# B&R Automation Studio project BaseProject (part 2)

### TrackMod.vvm - PC/TrackModule/TrackMod.vvm
```iecst
VAR_CONFIG
	Cyclic#1.::gSampleTrak AT %Q.TrackModule::TrackInterface.SampleTrak; (*Insert your comment here...*)
	Cyclic#1.TrackModule::gTrackModule AT %Q.TrackModule::TrackInterface.ModulePml; (*Insert your comment here...*)
	Cyclic#1.TrackModule::gAlarmXCore_TrackModule AT %Q.TrackModule::TrackInterface.AlarmCore; (*Insert your comment here...*)
	Cyclic#1.TrackModule::gRecipeXml_TrackModule AT %Q.TrackModule::TrackInterface.RecipeCore; (*Insert your comment here...*)
END_VAR
```

### TrakALM.mpalarmxcore - PC/TrackModule/mappServices/TrakALM.mpalarmxcore
```
Element gAlarmXCore_TrackModule (Type=mpalarmxcore)
  mapp.AlarmX.Core:
    Mapping:
      [0]:
        Alarm = Inf*
        [0] = Aggregate
          Name = TrakModuleInfo
      [1]:
        Alarm = Warn*
        [0] = Aggregate
          Name = TrakModuleWarning
      [2]:
        Alarm = Alrm*
        [0] = Aggregate
          Name = TrakModuleAlarm
    Default:
      [0] = Reaction
        Name = TrakTest
      [1] = Remain
  mapp.AlarmX.Core.Configuration:
    [0]:
      Name = Alrm_ErrorStop
      Message = {$TrakAssembly/TrakErrorStop}
      Code = 1000
      Behavior = DiscreteValueMonitoring
        Monitoring:
          MonitoredPV = TrakModule::AsmSampleT:fbAsmReadStatus.AssemblyErrorStop
          TriggerValues:
            [0] = TRUE
    [1]:
      Name = Inf_PowerOn
      Message = {$Assembly/Info/TrakPowerOn}
      Behavior = DiscreteValueMonitoring
        Monitoring:
          MonitoredPV = TrakModule::AsmSampleT:fbAsmReadInfo.AssemblyInfo.PowerOn
          TriggerValues:
            [0] = TRUE
    [2]:
      Name = Inf_ModuleTest
      Message = {$TrakAssembly/LocalTrakModuleInfo}
      Severity = 0
      Behavior = DiscreteValueMonitoring
        Monitoring:
          MonitoredPV = TrakModule::AsmAlarm:TriggerTestInformation
          TriggerValues:
            [0] = TRUE
    [3]:
      Name = Warn_ModuleTest
      Message = {$TrakAssembly/LocalTrakModuleWarning}
      Code = 100
      Severity = 50
      Behavior = DiscreteValueMonitoring
        Monitoring:
          MonitoredPV = TrakModule::AsmAlarm:TriggerTestWarning
          TriggerValues:
            [0] = TRUE
    [4]:
      Name = Alrm_ModuleTest
      Message = {$TrakAssembly/LocalTrakModuleAlarm}
      Code = 1000
      Severity = 100
      Behavior = DiscreteValueMonitoring
        Monitoring:
          MonitoredPV = TrakModule::AsmAlarm:TriggerTestAlarm
          TriggerValues:
            [0] = TRUE
    [5]:
      Name = TrakModuleInfo
      Message = {$TrakAssembly/Module.Info}
      AdditionalInformation1 = trakAlarmContent
    [6]:
      Name = TrakModuleWarning
      Message = {$TrakAssembly/Module.Warning}
      Code = 100
      AdditionalInformation1 = trakAlarmContent
    [7]:
      Name = TrakModuleAlarm
      Message = {$TrakAssembly/Module.Alarm}
      Code = 1000
      AdditionalInformation1 = trakAlarmContent
  mapp.AlarmX.Core.Snippets:
    [0]:
      Key = ModuleName
      Value:
        PV = TrakModule::ModuleName
  mapp.AlarmX.Core.Categories:
    [0]:
      Name = Information
      SourceProperty:
        Severity = 0..99
    [1]:
      Name = Warning
      SourceProperty:
        Severity = 100..199
    [2]:
      Name = Alarm
      SourceProperty:
        Severity = 1000..1199
```

### TrakMod.vvm - PC/TrakMod/TrakMod.vvm
```iecst
VAR_CONFIG
	Cyclic#1.::gSampleTrak AT %Q.Cyclic#1.TrakMod::TrakInterface.SampleTrak; (*Insert your comment here...*)
	Cyclic#1.TrakMod::gTrakModule AT %Q.Cyclic#1.TrakMod::TrakInterface.ModulePml; (*Insert your comment here...*)
	Cyclic#1.TrakMod::gAlarmXCore_TrakModule AT %Q.Cyclic#1.TrakMod::TrakInterface.AlarmCore; (*Insert your comment here...*)
	Cyclic#1.TrakMod::gRecipeXml_TrakModule AT %Q.Cyclic#1.TrakMod::TrakInterface.RecipeCore; (*Insert your comment here...*)
	Cyclic#1.::gSampleTrak_SectorTrakAll AT %Q.Cyclic#1.TrakMod::TrakInterface.SectorTrakAll; (*Insert your comment here...*)
	Cyclic#1.::gSampleTrak_SectorTrakB AT %Q.Cyclic#1.TrakMod::TrakInterface.SectorTrakB; (*Insert your comment here...*)
	Cyclic#1.::gSampleTrak_SectorTrakA AT %Q.Cyclic#1.TrakMod::TrakInterface.SectorTrakA; (*Insert your comment here...*)
END_VAR
```

### TrakALM.mpalarmxcore - PC/TrakMod/mappServices/TrakALM.mpalarmxcore
```
Element gAlarmXCore_TrakModule (Type=mpalarmxcore)
  mapp.AlarmX.Core:
    Mapping:
      [0]:
        Alarm = Inf*
        [0] = Aggregate
          Name = TrakModuleInfo
      [1]:
        Alarm = Warn*
        [0] = Aggregate
          Name = TrakModuleWarning
      [2]:
        Alarm = Alrm*
        [0] = Aggregate
          Name = TrakModuleAlarm
    Default:
      [0] = Remain
      [1] = Reaction
        Name = TrakTest
  mapp.AlarmX.Core.Configuration:
    [0]:
      Name = Alrm_ErrorStop
      Message = {$TrakAssembly/TrakErrorStop}
      Code = 1000
      Behavior = DiscreteValueMonitoring
        Monitoring:
          MonitoredPV = TrakMod::AsmSampleT:fbAsmReadStatus.AssemblyErrorStop
          TriggerValues:
            [0] = TRUE
    [1]:
      Name = Inf_PowerOn
      Message = {$TrakAssembly/TrakPowerOn}
      Behavior = DiscreteValueMonitoring
        Monitoring:
          MonitoredPV = TrakMod::AsmSampleT:fbAsmReadInfo.AssemblyInfo.PowerOn
          TriggerValues:
            [0] = TRUE
    [2]:
      Name = Inf_ModuleTest
      Message = {$TrakAssembly/LocalTrakModuleInfo}
      Severity = 0
      Behavior = DiscreteValueMonitoring
        Monitoring:
          MonitoredPV = TrakMod::AsmAlarm:TriggerTestInformation
          TriggerValues:
            [0] = TRUE
    [3]:
      Name = Warn_ModuleTest
      Message = {$TrakAssembly/LocalTrakModuleWarning}
      Code = 100
      Severity = 50
      Behavior = DiscreteValueMonitoring
        Monitoring:
          MonitoredPV = TrakMod::AsmAlarm:TriggerTestWarning
          TriggerValues:
            [0] = TRUE
    [4]:
      Name = Alrm_ModuleTest
      Message = {$TrakAssembly/LocalTrakModuleAlarm}
      Code = 1000
      Severity = 100
      Behavior = DiscreteValueMonitoring
        Monitoring:
          MonitoredPV = TrakMod::AsmAlarm:TriggerTestAlarm
          TriggerValues:
            [0] = TRUE
    [5]:
      Name = TrakModuleInfo
      Message = {$TrakAssembly/Module.Info}
      AdditionalInformation1 = trakAlarmContent
    [6]:
      Name = TrakModuleWarning
      Message = {$TrakAssembly/Module.Warning}
      Code = 100
      AdditionalInformation1 = trakAlarmContent
    [7]:
      Name = TrakModuleAlarm
      Message = {$TrakAssembly/Module.Alarm}
      Code = 1000
      AdditionalInformation1 = trakAlarmContent
  mapp.AlarmX.Core.Snippets:
    [0]:
      Key = ModuleName
      Value:
        PV = TrakMod::ModuleName
  mapp.AlarmX.Core.Categories:
    [0]:
      Name = Information
      SourceProperty:
        Severity = 0..99
    [1]:
      Name = Warning
      SourceProperty:
        Severity = 100..199
    [2]:
      Name = Alarm
      SourceProperty:
        Severity = 1000..1199
```

### TrakCFG.mprecipexml - PC/TrakMod/mappServices/TrakCFG.mprecipexml
```
Element gRecipeXml_TrakModule (Type=mprecipexml)
  Alarms = MpAlarmX
```

### TrakPML.mppackmlmodule - PC/TrakMod/mappServices/TrakPML.mppackmlmodule
```
Element gTrakModule (Type=mppackmlmodule)
  Module:
    Name = TrakAssembly
    Parent:
      Parent = gMainModule
      Activation = 0
```

### TrakModule.vvm - PC/TrakModule/TrakModule.vvm
```iecst
VAR_CONFIG
	Cyclic#1.::gSampleTrak AT %Q.TrakModule::TrakInterface.SampleTrak; (*Insert your comment here...*)
	Cyclic#1.TrakModule::gTrakModule AT %Q.TrakModule::TrakInterface.ModulePml; (*Insert your comment here...*)
	Cyclic#1.TrakModule::gAlarmXCore_TrakModule AT %Q.TrakModule::TrakInterface.AlarmCore; (*Insert your comment here...*)
	Cyclic#1.TrakModule::gRecipeXml_TrackModule AT %Q.TrakModule::TrakInterface.RecipeCore; (*Insert your comment here...*)
END_VAR
```

### TrakALM.mpalarmxcore - PC/TrakModule/mappServices/TrakALM.mpalarmxcore
```
Element gAlarmXCore_TrakModule (Type=mpalarmxcore)
  mapp.AlarmX.Core:
    Mapping:
      [0]:
        Alarm = Inf*
        [0] = Aggregate
          Name = TrakModuleInfo
      [1]:
        Alarm = Warn*
        [0] = Aggregate
          Name = TrakModuleWarning
      [2]:
        Alarm = Alrm*
        [0] = Aggregate
          Name = TrakModuleAlarm
    Default:
      [0] = Reaction
        Name = TrakTest
      [1] = Remain
  mapp.AlarmX.Core.Configuration:
    [0]:
      Name = Alrm_ErrorStop
      Message = {$TrakAssembly/TrakErrorStop}
      Code = 1000
      Behavior = DiscreteValueMonitoring
        Monitoring:
          MonitoredPV = TrakModule::AsmSampleT:fbAsmReadStatus.AssemblyErrorStop
          TriggerValues:
            [0] = TRUE
    [1]:
      Name = Inf_PowerOn
      Message = {$Assembly/Info/TrakPowerOn}
      Behavior = DiscreteValueMonitoring
        Monitoring:
          MonitoredPV = TrakModule::AsmSampleT:fbAsmReadInfo.AssemblyInfo.PowerOn
          TriggerValues:
            [0] = TRUE
    [2]:
      Name = Inf_ModuleTest
      Message = {$TrakAssembly/LocalTrakModuleInfo}
      Severity = 0
      Behavior = DiscreteValueMonitoring
        Monitoring:
          MonitoredPV = TrakModule::AsmAlarm:TriggerTestInformation
          TriggerValues:
            [0] = TRUE
    [3]:
      Name = Warn_ModuleTest
      Message = {$TrakAssembly/LocalTrakModuleWarning}
      Code = 100
      Severity = 50
      Behavior = DiscreteValueMonitoring
        Monitoring:
          MonitoredPV = TrakModule::AsmAlarm:TriggerTestWarning
          TriggerValues:
            [0] = TRUE
    [4]:
      Name = Alrm_ModuleTest
      Message = {$TrakAssembly/LocalTrakModuleAlarm}
      Code = 1000
      Severity = 100
      Behavior = DiscreteValueMonitoring
        Monitoring:
          MonitoredPV = TrakModule::AsmAlarm:TriggerTestAlarm
          TriggerValues:
            [0] = TRUE
    [5]:
      Name = TrakModuleInfo
      Message = {$TrakAssembly/Module.Info}
      AdditionalInformation1 = trakAlarmContent
    [6]:
      Name = TrakModuleWarning
      Message = {$TrakAssembly/Module.Warning}
      Code = 100
      AdditionalInformation1 = trakAlarmContent
    [7]:
      Name = TrakModuleAlarm
      Message = {$TrakAssembly/Module.Alarm}
      Code = 1000
      AdditionalInformation1 = trakAlarmContent
  mapp.AlarmX.Core.Snippets:
    [0]:
      Key = ModuleName
      Value:
        PV = TrakModule::ModuleName
  mapp.AlarmX.Core.Categories:
    [0]:
      Name = Information
      SourceProperty:
        Severity = 0..99
    [1]:
      Name = Warning
      SourceProperty:
        Severity = 100..199
    [2]:
      Name = Alarm
      SourceProperty:
        Severity = 1000..1199
```

### TrakCFG.mprecipexml - PC/TrakModule/mappServices/TrakCFG.mprecipexml
```
Element gRecipeXml_TrackModule (Type=mprecipexml)
  Alarms = MpAlarmX
```

### LoggerCFG.mappmotioncfg - PC/mappMotion/LoggerCFG.mappmotioncfg
```
Element MappMotionConfiguration (Type=mappmotioncfg)
  Logger:
    SelectiveLogging = Used
      AdministrativeCommands = Selective
      MovementCommands = Selective
      InformationalCommands = Selective
```

### AsmCfg.assembly - PC/mappMotion/TrakConfig/AsmCfg.assembly
```
Element gSampleTrak (Type=assembly)
  Tracks:
    TrackSeparation = 0.030
    Track[1]:
      Segments:
        SegmentRef[1] = ::gSeg_A_1
        SegmentRef[2] = ::gSeg_A_2
        SegmentRef[3] = ::gSeg_A_3
        SegmentRef[4] = ::gSeg_A_4
        SegmentRef[5] = ::gSeg_A_5
        SegmentRef[6] = ::gSeg_A_6
        SegmentRef[7] = ::gSeg_A_7
        SegmentRef[8] = ::gSeg_A_8
        SegmentRef[9] = ::gSeg_A_9
        SegmentRef[10] = ::gSeg_A_10
        SegmentRef[11] = ::gSeg_A_11
        SegmentRef[12] = ::gSeg_A_12
      Position = Absolute
        SegmentRef = ::gSeg_A_1
        SegmentCountDirection = RightToLeft
        Translation:
          X = 0.0
          Y = 0.0
          Z = 0.0
        Orientation:
          Angle1 = 0.0
          Angle2 = 0.0
          Angle3 = 180
  CommonSegmentSettings:
    SegmentSimulationOnPLC = Off
    StopReaction = InductionHalt
    SpeedFilter = NotUsed
    ControllerParameters:
      DefaultParameter:
        Controller:
          Position:
            ProportionalGain = 200
          Speed:
            ProportionalGain = 80
            IntegrationTime = 0.0
          FeedForward:
            TotalMass = 1
            ForcePositive = 0.0
            ForceNegative = 0.0
            SpeedForceFactor = 0.0
            ForceLoad = 0.0
        MovementErrorLimits:
          PositionError = 0.001
          VelocityError = 0.05
      AdditionalParameterSets = NotUsed
    ScopeOfErrorReaction = Assembly
    ShuttleIdentificationTime = 0
  Shuttles:
    MaxShuttleCount = 150
    DistanceReserve:
      Collision = 0.002
      ErrorStop = 0.006
    ShuttleStereotypes:
      ShuttleStRef[1] = gSampleShuttle
    MagnetPlateConfigurations:
      ShuttleType[1] = 8F1SA.100.xxxxxx-x
    CollisionAvoidance:
      Strategy = Constant
      MaximumModelDimensions:
        Length:
          ExtentToFront = 0.025
          ExtentToBack = 0.025
        Width:
          Width = 0.040
  AssemblyFeatures:
    AssemblyFeatureRef[1] = SampleTrak_AutoAttach
    AssemblyFeatureRef[2] = SampleTrak_LocalLimits
    AssemblyFeatureRef[3] = SampleTrak_SimShuttle
  Visualization:
    MonitoringPv = gSampleTrakMon
    ProcessingTaskClass = 1
```

### AsmFeatCfg.assemblyfeature - PC/mappMotion/TrakConfig/AsmFeatCfg.assemblyfeature
```
Element SampleTrak_AutoAttach (Type=assemblyfeature)
  Type = ShtSectorAutoAttach
    Priority[1]:
      SectorRef = SampleTrak_SectorTrackA
      Orientation = KeepSegment
Element SampleTrak_LocalLimits (Type=assemblyfeature)
  Type = LocalLimits
    LocalLimit[1]:
      Location:
        SectorRef = SampleTrak_SectorTrackA
      MotionLimits:
        Velocity = Basic
          Velocity = 3
        Acceleration = Basic
          Acceleration = 10
Element SampleTrak_SimShuttle (Type=assemblyfeature)
  Type = InitShuttleSim
    InitShuttleSim[1]:
      SectorRef = SampleTrak_SectorTrackA
      Orientation = Positive
      ShuttleDefinition = ShuttleSetDefinition
        StartPosition = 0.0
        NumberOfShuttles = 10
        DistnaceBetweenShuttles = 100
Element SampleTrak_AsmPwr_STO1 (Type=assemblyfeature)
  Type = ExcludeFromAssembly
    Exclusion = AsmPowerOn
      SegmentRef[1] = ::Seg_A_1
      SegmentRef[2] = ::Seg_A_2
Element SampleTrak_AsmPwr_STO2 (Type=assemblyfeature)
  Type = ExcludeFromAssembly
    Exclusion = AsmPowerOn
      SegmentRef[1] = ::Seg_A_3
      SegmentRef[2] = ::Seg_A_4
```

### SectorCfg.sector - PC/mappMotion/TrakConfig/SectorCfg.sector
```
Element gSampleTrak_SectorTrakA (Type=sector)
  Type = Composed
    StartSegment:
      SegmentRef = ::gSeg_A_1
    IntermediateSegments:
      SegmentRef[1] = ::gSeg_A_2
      SegmentRef[2] = ::gSeg_A_3
      SegmentRef[3] = ::gSeg_A_4
      SegmentRef[4] = ::gSeg_A_5
      SegmentRef[5] = ::gSeg_A_6
      SegmentRef[6] = ::gSeg_A_7
      SegmentRef[7] = ::gSeg_A_8
      SegmentRef[8] = ::gSeg_A_9
      SegmentRef[9] = ::gSeg_A_10
      SegmentRef[10] = ::gSeg_A_11
    EndSegment:
      SegmentRef = ::gSeg_A_12
      PositionRelativeTo = FromEnd
```

### ShuttleCfg.shuttlestereotype - PC/mappMotion/TrakConfig/ShuttleCfg.shuttlestereotype
```
Element SampleShuttle (Type=shuttlestereotype)
  MeasurementUnit = 5067858
  MeasurementResolution = 0.00001
  MovementLimits = Internal
    VelocityIsReadOnly = 0
    Velocity:
      Velocity = 4
    AccelerationIsReadOnly = 0
    Acceleration:
      Acceleration = 40
    DecelerationIsReadOnly = 0
    Deceleration:
      Deceleration = 40
  JerkFilter = Used
    JerkTime = 0.02
  UserData:
    Size = 12
```

### MainAlrCfg.mpalarmxcore - PC/mappServices/Alarm/MainAlrCfg.mpalarmxcore
```
Element gAlarmXCore (Type=mpalarmxcore)
  mapp.AlarmX.Core:
    Mapping:
      [0]
  mapp.AlarmX.Core.Configuration:
    [0]:
      Name = MainTestAlarm
      Message = This is just a test for main
      Behavior = DiscreteValueMonitoring
        Monitoring:
          MonitoredPV = ::TSMAlarm:TriggerTestAlarm
          TriggerValues:
            [0] = TRUE
```

### AuditCfg.mpaudittrail - PC/mappServices/Diagnostic/AuditCfg.mpaudittrail
```
Element gAuditTrail (Type=mpaudittrail)
  Audit:
    Events:
      [0] = 18
    TextSource:
      OutputFormat = {&typ} | {&msg} | {&cmt}
  Alarms = MpAlarmX
```

### MachCfg.mprecipexml - PC/mappServices/MachineConfig/MachCfg.mprecipexml
```
Element gRecipeXml (Type=mprecipexml)
  Alarms = MpAlarmX
```

### Main.mppackmlmodule - PC/mappServices/Operation/Main.mppackmlmodule
```
Element gMainModule (Type=mppackmlmodule)
  Module:
    Parent = 1
      Unit = gPackMLCore
      Activation = 0
```

## Logical view

Binary libraries used (declarations not repeated): operator, runtime, astime, AsIecCon, AsZip, FileIO, sys_lib, snprintf 1.10.2, brdkSTR, ArEventLog, AsHttp, AsIODiag, AsBrStr, standard, asstring, McBase 5.15.1, McAcpPar 5.15.1, McAxGroup 5.15.1, McAcpAx 5.15.1, McAxis 5.15.1, McPathGen 5.15.1, McProgInt 5.15.1, McAcpTrak 5.15.1, MpRobotics 5.15.1, MpAxis 5.15.1, MpBase 5.15.0, MpCom 5.14.0, MpPackML 5.15.0, MpFile 5.15.0, MpAudit 5.15.0, MpRecipe 5.15.0, MpAlarmX 5.15.0, CoTrace 5.15.0, MpServer 5.15.0

### Global.typ - Global data types
```iecst
TYPE
	ShuttleUserDataType : 	STRUCT  (*Shuttle data type definition - application specific*)
		ID : UINT; (*Shuttle ID assigned during homing*)
	END_STRUCT;
	SubroutineSequenceType : 	STRUCT  (*Subroutine sequence structure for a module*)
		Cmd : SubroutineSequenceCommandType; (*Subroutine commands (inputs)*)
		Status : SubroutineSequenceStatusType; (*Subroutine statuses (outputs)*)
	END_STRUCT;
	SubroutineSequenceCommandType : 	STRUCT  (*Subroutine seguence command variables*)
		Start : BOOL; (*Initiate the subroutine execution when the status reports ready*)
		Stop : BOOL; (*If the main routine is no longer in a proper state to execute the subroutine, stop the subroutine*)
		ErrorReset : BOOL; (*Command to reset the subroutine if in error*)
	END_STRUCT;
	SubroutineSequenceStatusType : 	STRUCT  (*Subroutine segeuqnce status variables*)
		Ready : BOOL; (*The subroutine is ready to start*)
		Complete : BOOL; (*The subroutine has complete and will wait for the reset of the start command*)
		Error : BOOL; (*The subroutine is in error and needs to be reset*)
	END_STRUCT;
	CyclicSubroutineType : 	STRUCT  (*Cyclic subroutine structure definition for a module*)
		Cmd : CyclicSubroutineCommandType; (*Cyclic subroutine command structure*)
		Status : CyclicSubroutineStatusType; (*Cyclic subroutine status structure*)
	END_STRUCT;
	CyclicSubroutineCommandType : 	STRUCT  (*Cyclic subroutine command structure definition*)
		Activate : BOOL; (*Activate the subroutine cyclic operation*)
		ErrorReset : BOOL; (*Reset the subroutine when in error*)
	END_STRUCT;
	CyclicSubroutineStatusType : 	STRUCT  (*Cyclic subroutine status structure definition*)
		Ready : BOOL; (*The subroutine cyclic operation is ready to begin*)
		Active : BOOL; (*The subroutine is activated and running*)
		Error : BOOL; (*The subroutine is in error*)
	END_STRUCT;
END_TYPE

(*Trak Data Datatypes*)
```

### Global.var - Global variables
```iecst
VAR
	gTrakData : TrkDiagStatusType;
END_VAR
```

### Package Logical/Libraries - Global libraries

### Library Logical/Libraries/TrBase (IEC) - AddOn Trak library for types and variable definitions

#### TrBase.typ - Exported data types
```iecst
(*Assembly States*)

TYPE
	TrBaseAsmStateEnum :
		(
		ASM_STATE_OFF := 0,
		ASM_STATE_POWER,
		ASM_STATE_INIT,
		ASM_STATE_READY,
		ASM_STATE_ERROR := 255
		);
END_TYPE

(*Assembly Control*)

TYPE
	TrBaseAsmType : 	STRUCT
		Cmd : TrBaseAsmCmdType;
		Status : TrBaseAsmStatusType;
	END_STRUCT;
END_TYPE

(*Assembly Command*)

TYPE
	TrBaseAsmCmdType : 	STRUCT
		Power : BOOL; (*Switch on all segment controllers and identify all shuttles. Requires AssemblyDisabled.*)
		Stop : BOOL; (*Stop all shuttles and switch off all segment controllers*)
		ErrorReset : BOOL; (*Reset the assembly if Assembly FB error or AssemblyErrorStop*)
	END_STRUCT;
END_TYPE

(*Assembly Status*)

TYPE
	TrBaseAsmStatusType : 	STRUCT
		Disabled : BOOL; (*[mapp Trak] The assembly is switched off. AsmPowerOff.Done, AsmReset.Done, or power cycle*)
		Homing : BOOL; (*[mapp Trak] Shuttle identification is active. AsmPowerOn.Execute*)
		Ready : BOOL; (*[mapp Trak] The assembly is switched on. AsmPowerOn.Done*)
		Stopping : BOOL; (*[mapp Trak] The shuttles are stopped. AsmPowerOff.Execute*)
		ErrorStop : BOOL; (*[mapp Trak] The shuttles are stopped. An error has occured in the assembly*)
		CommunicationReady : BOOL; (*[mapp Trak] The network of all segments has been initialized*)
		ReadyForPowerOn : BOOL; (*[mapp Trak] All segment controllers are ready to be switched on*)
		PowerOn : BOOL; (*[mapp Trak] All segments are switched on*)
		StartupCount : UDINT; (*[mapp Trak] Number of assembly switch-on operations*)
		ShuttlesInErrorStopCount : UINT; (*[mapp Trak] Number of shuttles in state ErrorStop*)
		Error : BOOL; (*The assembly implementation is in error*)
	END_STRUCT;
	TrBaseTrackingCmdType : 	STRUCT
		Delete : BOOL;
	END_STRUCT;
	TrBaseTrackingStatusType : 	STRUCT
		ShuttlesToBeDeletedCount : DINT;
	END_STRUCT;
	TrBaseTrackingType : 	STRUCT
		Cmd : TrBaseTrackingCmdType;
		Status : TrBaseTrackingStatusType;
	END_STRUCT;
END_TYPE
```

#### TrBaseAlarm.typ - Exported data types
```iecst
TYPE
	TrBaseAlarmEnum :
		(
		trBASE_ALM_CONFIG_SAVE_FAILED,
		trBASE_ALM_CONFIG_LOAD_FAILED
		);
END_TYPE
```

#### TrBaseError.typ - Exported data types
```iecst
TYPE
	TrBaseErrorCodeEnum :
		(
		trBASE_NO_ERROR := 0, (*No Error*)
		trBASE_WRN_SAMPLE := -1609957375,
		trBASE_ERR_SAMPLE := -536215551
		);
END_TYPE
```

#### TrBase.fun - Exported functions and function blocks
```iecst
{REDUND_ERROR} FUNCTION TrBaseAddShToBuffer : UDINT (*Placeholder*) (*$GROUP=User,$CAT=User,$GROUPICON=User.png,$CATICON=User.png*)
	VAR_INPUT
		Axis : McAxisType;
		ShuttleBuffer : UDINT;
		BufferSize : UINT;
	END_VAR
END_FUNCTION

{REDUND_ERROR} FUNCTION TrBaseClearShBuffer : UDINT (*Placeholder*) (*$GROUP=User,$CAT=User,$GROUPICON=User.png,$CATICON=User.png*)
	VAR_INPUT
		ShuttleBuffer : UDINT;
		BufferSize : UINT;
	END_VAR
END_FUNCTION
```

#### TrBaseClearShBuffer.st
```iecst
(* Placeholder *)
FUNCTION TrBaseClearShBuffer

		ShuttleBuffer;
		BufferSize;

		TrBaseClearShBuffer := 0;

END_FUNCTION

(* Placeholder *)
FUNCTION TrBaseAddShToBuffer

		Axis;
		ShuttleBuffer;
		BufferSize;

		TrBaseAddShToBuffer := 0;
END_FUNCTION
```

### Library Logical/Libraries/TrkDiag (ANSIC)

#### TrkDiag.typ - Exported data types
```iecst
TYPE
	TrkDiagSegStatusDCBusType : 	STRUCT
		DCBusVoltage : REAL;
		DCBusVoltageMax : REAL;
		DCBusVoltageMin : REAL;
	END_STRUCT;
END_TYPE

(*Temporary Segment information*)

TYPE
	TrkDiagSegStatusTempType : 	STRUCT
		TemperatureCON : REAL; (*monitor temperature CON*)
		TemperaturePROZ : REAL; (*monitor temperature PROZ*)
		TemperatureAIR : REAL; (*monitor temperature AIR*)
		TemperatureBAL : REAL; (*monitor temperature BAL*)
		TemperatureCHASSIS_1 : REAL; (*monitor temperature CHASSIS_1*)
		TemperatureCHASSIS_2 : REAL; (*monitor temperature CHASSIS_2*)
		TemperatureCHASSIS_3 : REAL; (*monitor temperature CHASSIS_3*)
		TemperaturePOWER_SENS3 : REAL; (*monitor temperature POWER_SENS3*)
		TemperaturePOWER_SENS4 : REAL; (*monitor temperature POWER_SENS4*)
		TemperaturePOWER_SENS5 : REAL; (*monitor temperature POWER_SENS5*)
		TemperaturePOWER_SENS6 : REAL; (*monitor temperature POWER_SENS6*)
		TemperaturePOWER_SENS7 : REAL; (*monitor temperature POWER_SENS7*)
		TemperaturePOWER_SENS8 : REAL; (*monitor temperature POWER_SENS8*)
		TemperaturePOWER_SENS9 : REAL; (*monitor temperature POWER_SENS9*)
		TemperaturePOWER_SENS10 : REAL; (*monitor temperature POWER_SENS10*)
		TemperaturePOWER_SENS11 : REAL; (*monitor temperature POWER_SENS11*)
	END_STRUCT;
END_TYPE
```

#### TrkDiag.fun - Exported functions and function blocks
```iecst
FUNCTION_BLOCK tdSystemMonitorFb
	VAR
		Enable : USINT;
		New_Member5 : USINT;
		New_Member4 : USINT;
		New_Member3 : USINT;
		New_Member2 : USINT;
		New_Member1 : USINT;
		New_Member : USINT;
	END_VAR
END_FUNCTION_BLOCK
```

### Library Logical/Libraries/TrkPaper (ANSIC)
Depends on: McAcpTrak, snprintf, brdkSTR, TrkDiag

#### TrkPaper.typ - Exported data types
```iecst
(*Trak Master Core Types*)

TYPE
	TrkPaperCoreAxisLookupType : 	STRUCT  (*Lookup table datatype*)
		Present : BOOL; (*Axis is present and a valid reference exists*)
		Axis : McAxisType; (*Axis information*)
	END_STRUCT;
	TrkPaperCoreColorOffsetsType : 	STRUCT  (*Userdata color offsets*)
		Red : UDINT; (*Offset for UserData address for the Red color in USINT*)
		Green : UDINT; (*Offset for UserData address for the Green color in USINT*)
		Blue : UDINT; (*Offset for UserData address for the Blue color in USINT*)
	END_STRUCT;
	TrkPaperCoreColorOptionType : 	STRUCT  (*Shuttle Color Option*)
		Enabled : BOOL; (*Option is enabled*)
		Offsets : TrkPaperCoreColorOffsetsType; (*Userdata color offsets*)
	END_STRUCT;
	TrkPaperCoreErrorEnum :
		( (*Error Enumeration*)
		trkPAPER_CORE_ERR_OK := 0, (*No error present*)
		trkPAPER_CORE_ERR_INVALID_ASM := -61000, (*Invalid input assembly reference*)
		trkPAPER_CORE_ERR_SH_CNT_EXCD := -61001, (*Maximum shuttle count exceeded. Need to increase max shuttle count constant*)
		trkPAPER_CORE_ERR_STR_LEN_EXCD := -61002 (*The built string is too long, need to increase the maximum size to prevent page faulting*)
		);
	TrkPaperCoreInternalType : 	STRUCT  (*Internal Datatype*)
		TypeID : UDINT; (*TypeID to help with handle application*)
		State : USINT; (*State of execution*)
	END_STRUCT;
	TrkPaperCoreOptionsType : 	STRUCT  (*Options for Core Function Block*)
		Color : TrkPaperCoreColorOptionType; (*Shuttle Color Option*)
		Shuttle : TrkPaperCoreShuttleOptionType; (*Shuttle Option*)
	END_STRUCT;
	TrkPaperCoreShuttleOptionType : 	STRUCT  (*Shuttle Option*)
		Enabled : BOOL; (*Option is enabled*)
	END_STRUCT;
	TrkPaperCoreStateEnum :
		( (*State of execution*)
		trkPAPER_CORE_OFF, (*Waiting for enable command*)
		trkPAPER_CORE_INIT, (*Initialization state*)
		trkPAPER_CORE_RUNNING, (*Running state*)
		trkPAPER_CORE_RESET, (*Resetting state*)
		trkPAPER_CORE_ERROR (*Error state*)
		);
	TrkPaperCoreSvgLengthsType : 	STRUCT  (*String lengths of SVGs*)
		ContentLength : UDINT; (*String Length of SVG Content string*)
		TransformLength : UDINT; (*String Length of SVG Transform string*)
	END_STRUCT;
	TrkPaperCoreViewBoxCfgType : 	STRUCT  (*Attributes of the SVG's viewbox*)
		MinX : REAL; (*Minimum x position*)
		MinY : REAL; (*minimum y position*)
		Width : REAL; (*Width of viewbox*)
		Height : REAL; (*Height of viewbox*)
	END_STRUCT;
	TrkPaperSegmentStyleEnumeration :
		( (*Style enumeration for the trak map strings*)
		trkPAPER_SEG_STYLE_DEFAULT := 0, (*Segment Default Style*)
		trkPAPER_SEG_STYLE_ERROR := 1, (*Segment is in error style*)
		trkPAPER_SEG_STYLE_OKAY := 2, (*Segment is okay style*)
		trkPAPER_SEG_STYLE_WARNING := 3 (*Segment is in a warning state style*)
		);
	TrkPaperShuttleControlErrorEnum :
		( (*Error enumeration*)
		trkPAPER_SH_CTRL_ERR_OK := 0, (*No error currently*)
		trkPAPER_SH_CTRL_WARN_SH_NOT_AVA := -52000, (*Shuttle Currently not listed as available*)
		trkPAPER_SH_CTRL_WARN_NO_ELEM_FN := -52001, (*Input selected element did not return a shuttle*)
		trkPAPER_SH_CTRL_ERR_INVALID_HDL := -62000, (*Invalid input handle*)
		trkPAPER_SH_CTRL_ERR_EL_MOVE := -62001 (*Error in an elastic movment*)
		);
	TrkPaperShuttleControlFbType : 	STRUCT  (*Internal Function Blocks*)
		ShGetInfo : MC_BR_ShReadInfo_AcpTrak; (*Shuttle Get info*)
		ElMoveAbs : MC_BR_ElasticMoveAbs_AcpTrak; (*Elastic move absolute command*)
		ElMoveAdd : MC_BR_ElasticMoveAdd_AcpTrak; (*Elastic move addtive command*)
	END_STRUCT;
END_TYPE

(*Trak Master Shuttle Control Types*)

TYPE
	TrkPaperShuttleControlParsType : 	STRUCT  (*Input parameters for Shuttle Control*)
		Position : LREAL; (*Destination position for Absolute and Velocity commands*)
		Distance : LREAL; (*Distance for all relative commands*)
		Vel : REAL; (*Comanded Movement velocity*)
		Accel : REAL; (*Comanded Movement acceleration*)
		Decel : REAL; (*Comanded Movement deceleration*)
	END_STRUCT;
	TrkPaperShuttleControlStatesEnum :
		( (*State of execution*)
		trkPAPER_SH_CONTROL_OFF, (*Off State*)
		trkPAPER_SH_CONTROL_INIT, (*Init/Waiting for valid ShElement state*)
		trkPAPER_SH_CONTROL_IDLE, (*Idle waiting for a command state*)
		trkPAPER_SH_CONTROL_EL_MOVE_ABS, (*Move Elastic absoulte active state*)
		trkPAPER_SH_CONTROL_EL_MOVE_ADD, (*Move Elastic Additive active state*)
		trkPAPER_SH_CONTROL_MOVE_DONE, (*Move has completed*)
		trkPAPER_SH_CONTROL_ERROR (*Error present on the FB*)
		);
	TrkPaperShuttleCtrlInternalType : 	STRUCT  (*Internal data type*)
		State : TrkPaperShuttleControlStatesEnum; (*State of execution*)
		CoreInt : REFERENCE TO TrkPaperCoreInternalType; (*Internal data for the Core function block*)
		CurrentAxis : McAxisType; (*Current selected Axis*)
		Fbs : TrkPaperShuttleControlFbType; (*Internal function blocks*)
		Idx : USINT; (*Selected Index for the axis lookup table*)
		LastIdx : USINT; (*Last cycle selected index for the axis lookup table*)
	END_STRUCT;
END_TYPE
```

#### TrkPaper.var - Exported constants
```iecst
VAR CONSTANT
	trkPAPER_SEG_COLOR_OFFSET : UDINT := 4;
	trkPAPER_MAX_SHUTTLE_COUNT : USINT := 150;
	trkPAPER_MAX_SHUTLE_ARRAY : USINT := trkPAPER_MAX_SHUTTLE_COUNT-1;
	trkPAPER_CORE_CORE_TYPE_ID : DINT := 651684313;
	trkPAPER_CORE_MAX_STR_LEN : UDINT := 200000;
END_VAR
```

#### TrkPaper.fun - Exported functions and function blocks
```iecst
FUNCTION_BLOCK TrkPaperCore (*Core Trak Paper Function Block*)
	VAR_INPUT
		Enable : BOOL; (*Enables the core functionality*)
		ErrorRest : BOOL; (*Reset any present errors*)
		Assembly : REFERENCE TO McAssemblyType; (*Assembly reference to monitor*)
		ShuttleMon : REFERENCE TO McAcpTrakAssemblyMonData; (*Shuttle Monitor structure for the assembly*)
		Segments : REFERENCE TO TrkDiagSegmentType; (*Address of the segment list for the system*)
		SegmentCount : USINT; (*Count of the segments in the system*)
		ViewBoxCfg : TrkPaperCoreViewBoxCfgType; (*View box configuration for the SVG*)
		Options : REFERENCE TO TrkPaperCoreOptionsType; (*Options for the core fb*)
	END_VAR
	VAR_OUTPUT
		Error : BOOL; (*Error present on FB*)
		ErrorID : TrkPaperCoreErrorEnum; (*Error ID of current error*)
		Active : BOOL; (*Function block is active*)
		SvgTransform : STRING[trkPAPER_CORE_MAX_STR_LEN]; (*SVG Transform string to tie to a paper widget*)
		SvgContent : STRING[trkPAPER_CORE_MAX_STR_LEN]; (*SVG Content string to tie to a Paper widget*)
		StrLengths : TrkPaperCoreSvgLengthsType; (*Diagnostic viewer to see current lengths of SVG Content/Transform*)
		Handle : UDINT; (*Handle used for other Trak Master Function Blocks*)
	END_VAR
	VAR
		Internal : TrkPaperCoreInternalType; (*Internal data type*)
	END_VAR
END_FUNCTION_BLOCK

FUNCTION_BLOCK TrkPaperShuttleControl (*Shuttle Control Function Block*)
	VAR_INPUT
		Enable : BOOL; (*Enables the shuttle controller*)
		Handle : UDINT; (*Handle of the Core Trak Master Function Block*)
		SelectedElem : STRING[80]; (*Selected Element String that is populated from a Paper Widget*)
		ElasticMoveAbs : BOOL; (*Command to send shuttle on Elastic Move Absolute*)
		ElasticMoveAdd : BOOL; (*Command to send shuttle on Elastic Move Additive*)
		Parameters : REFERENCE TO TrkPaperShuttleControlParsType; (*Parameters for movement commands*)
	END_VAR
	VAR_OUTPUT
		Active : BOOL; (*Function block is currently Active*)
		MovementActive : BOOL; (*Controlled Shuttle is currently moving*)
		MovementDone : BOOL; (*Controlled Shuttle has completed movement*)
		Valid : BOOL; (*Input Selected Element is a valid controllable shuttle*)
		ShInfo : McAcpTrakShInfoType; (*Selected shuttle's current info. Only is Valid when Valid flag is set*)
		Error : BOOL; (*Error Present on FB*)
		ErrorID : DINT; (*Error ID of current Error*)
	END_VAR
	VAR
		Internal : TrkPaperShuttleCtrlInternalType; (*Internal data type*)
	END_VAR
END_FUNCTION_BLOCK

FUNCTION_BLOCK TrkPaperShuttleFeature (*Shuttle Feature Function Block*)
END_FUNCTION_BLOCK
```

#### TrkPaperCore.c
```c
#include <bur/plctypes.h>
#include <stdint.h>
#include <AsBrStr.h>

#define TRUE 1
#define FALSE 0

#ifdef __cplusplus
	extern "C"
	{
#endif
#include "TrkPaper.h"
#ifdef __cplusplus
	};
#endif

//Function Declaration to remove compiler warnings

//Verify that the two string lengths do not exceed a length
plcbit CheckStrLen(char* dest,char* source,UDINT length){
	if(brdkStrLen((uintptr_t)dest) + brdkStrLen((uintptr_t)source) >= length){
		return FALSE;
	}
	else{
		return TRUE;
	}
}

DINT StartSVGStrings(char* svgContent,
	char* svgTransform,
struct TrkPaperCoreViewBoxCfgType* viewBox){

	char tmp[150];

	brsmemset((uintptr_t)svgContent,0,sizeof(*svgContent));
	brsmemset((uintptr_t)svgTransform,0,sizeof(*svgTransform));

	snprintf2(tmp,150,"<svg viewBox=\"%f %f %f %f\">",
		viewBox->MinX,
		viewBox->MinY,
		viewBox->Width,
		viewBox->Height);
	if(CheckStrLen(svgContent,(char*)&tmp,trkPAPER_CORE_MAX_STR_LEN)){
		brsstrcat((uintptr_t)svgContent,(uintptr_t)&tmp);
	}
	else
		return trkPAPER_CORE_ERR_STR_LEN_EXCD;
	if(CheckStrLen(svgTransform,(char*)&"[",trkPAPER_CORE_MAX_STR_LEN)){
		brsstrcat((uintptr_t)svgTransform,(uintptr_t)&"[");
	}
	else
		return trkPAPER_CORE_ERR_STR_LEN_EXCD;
	//No Error, finished everything return OK
	return trkPAPER_CORE_ERR_OK;

}

//Closes the Transform and Content strings with the appropriate tags
DINT CloseSVGStrings(char* svgContent,
char* svgTransform){
	if(CheckStrLen(svgContent,(char*)&"</svg>",trkPAPER_CORE_MAX_STR_LEN)){
		brsstrcat((uintptr_t)svgContent,(uintptr_t)&"</svg>");
	}
	else
		return trkPAPER_CORE_ERR_STR_LEN_EXCD;
	if(CheckStrLen(svgTransform,(char*)&"]",trkPAPER_CORE_MAX_STR_LEN)){
		brsstrcat((uintptr_t)svgTransform,(uintptr_t)&"]");
	}
	else
		return trkPAPER_CORE_ERR_STR_LEN_EXCD;

	//No Error, finished everything return OK
	return trkPAPER_CORE_ERR_OK;
}

//Method for building the shuttle transform string. Defined the style of a segment based upon the information input into the FB
DINT BuildSegmentStrings(char* svgContent,
	char* svgTransform,
	struct TrkDiagSegmentType* segList,
USINT SegmentCount){

	USINT i;
	char tmp[200];

	//{"select":"#Segment","fill":1"}
	for (i = 0; i < SegmentCount; i++){
		if(segList[i].Status.ErrorCode > 0){
			snprintf2(tmp,200,"{\"select\":\"#%s\",\"style\":\"fill:%d\"}",
				segList[i].Name, //Segment Name
				trkPAPER_SEG_STYLE_ERROR //Segment Style Color index
				);

		}
		else if(!segList[i].Status.CommunicationReady || !segList[i].Status.ReadyForPowerOn){
			snprintf2(tmp,200,"{\"select\":\"#%s\",\"style\":\"fill:%d\"}",
				segList[i].Name, //Segment Name
				trkPAPER_SEG_STYLE_WARNING //Segment Style Color index
				);
		}
		else if(segList[i].Status.PowerOn){
			snprintf2(tmp,200,"{\"select\":\"#%s\",\"style\":\"fill:%d\"}",
				segList[i].Name, //Segment Name
				trkPAPER_SEG_STYLE_OKAY //Segment Style Color index
				);
		}
		else{
			snprintf2(tmp,200,"{\"select\":\"#%s\",\"style\":\"fill:%d\"}",
				segList[i].Name, //Segment Name
				trkPAPER_SEG_STYLE_DEFAULT //Segment Style Color index
				);
		}

		if(CheckStrLen(svgTransform,(char*)&tmp,trkPAPER_CORE_MAX_STR_LEN)){
			brsstrcat((uintptr_t)svgTransform,(uintptr_t)&tmp);
			if(CheckStrLen(svgTransform,(char*)&",",trkPAPER_CORE_MAX_STR_LEN)){
				//Every one except for the last index add a comma
				if(i != SegmentCount-1){
					brsstrcat((uintptr_t)svgTransform,(uintptr_t)&",");
				}
			}
			else{
				return trkPAPER_CORE_ERR_STR_LEN_EXCD;
			}

		}
		else
			return trkPAPER_CORE_ERR_STR_LEN_EXCD;
	}

	return trkPAPER_CORE_ERR_OK;

}

/* Core Trak Master function blocks. Handles the building of the SVG string */
void TrkPaperCore(struct TrkPaperCore* inst)
{
	switch (inst->Internal.State){
		case trkPAPER_CORE_OFF:
			//******************************************************************************** Off state
			if(inst->Enable){
				inst->Internal.TypeID = trkPAPER_CORE_CORE_TYPE_ID;
				inst->Handle = (uintptr_t)&inst->Internal;

				inst->Active = TRUE;
				inst->Internal.State = trkPAPER_CORE_INIT;
			}
			break;
		case trkPAPER_CORE_INIT:
			inst->Internal.State = trkPAPER_CORE_RUNNING;
			break;

		case trkPAPER_CORE_RUNNING:
			StartSVGStrings((char*)&inst->SvgContent,(char*)&inst->SvgTransform,&inst->ViewBoxCfg);

			inst->ErrorID = BuildSegmentStrings((char*)&inst->SvgContent,(char*)&inst->SvgTransform,inst->Segments,inst->SegmentCount);

			CloseSVGStrings((char*)&inst->SvgContent,(char*)&inst->SvgTransform);
			inst->StrLengths.ContentLength = brdkStrLen((uintptr_t)&inst->SvgContent);
			inst->StrLengths.TransformLength = brdkStrLen((uintptr_t)&inst->SvgTransform);

			if(inst->ErrorID != trkPAPER_CORE_ERR_OK){
				inst->Error = TRUE;

				inst->Internal.State = trkPAPER_CORE_ERROR;
			}
			if(!inst->Enable){
				inst->Active = FALSE;
				inst->Internal.State = trkPAPER_CORE_OFF;
			}
			break;
		case trkPAPER_CORE_RESET:
			//Try and recover by resetting any blocks

			break;
		case trkPAPER_CORE_ERROR:
			if(inst->ErrorRest){
				inst->Error = FALSE;
				inst->ErrorID = trkPAPER_CORE_ERR_OK;

				inst->Internal.State = trkPAPER_CORE_OFF;
			}
			break;
	}
}
```

#### TrkPaperShuttleControl.c
```c
#include <bur/plctypes.h>

#define TRUE 1
#define FALSE 0

#ifdef __cplusplus
	extern "C"
	{
#endif
#include "TrkPaper.h"
#ifdef __cplusplus
	};
#endif

plcbit CheckValidity(char* selectedElem){
	char buf[2];
	//Get a substring of the first 3 characters
	brdkStrSubStr(&buf,selectedElem,0,3);
	//Look at the start of the selectedID, if it starts with #ID then we know a shuttle has been clicked
	if(0 == brsstrcmp(&buf,&"#ID")){
		return TRUE;
	}
	else{
		return FALSE;
	}
}
USINT GetIndex(char* selectedElem){
	char buf[3];
	brdkStrSubStr(&buf,selectedElem,3,brdkStrLen(selectedElem) - 3);
	return (USINT)brdkStrAToUdint(&buf,BRDK_STR_CONVERT_DECIMAL);
}
/* Function block for handling a shuttle control provided from the paper element's selected element ID. Must be paired with the tmCore FB */
void TrkPaperShuttleControl(struct TrkPaperShuttleControl* inst)
{
	//TODO Code disabled for the moment as major type changes are occuring. Will need to revist at a future time.

//	if(inst->Valid){
//		inst->ShInfo = inst->Internal.Fbs.ShGetInfo.ShuttleInfo;
//	}
//	switch (inst->Internal.State){
//		case trkPAPER_SH_CONTROL_OFF:
//			//******************************************************************************** Off state
//			if(inst->Enable){
//				if(inst->Handle == 0){
//					inst->Error = TRUE;
//					inst->ErrorID = trkPAPER_SH_CONTROL_ERR_INVALID_HANDLE;
//
//					inst->Internal.State = trkPAPER_SH_CONTROL_ERROR;
//				}
//				else{
//					inst->Internal.CoreInt = (TpCoreInternalTyp*)inst->Handle;
//					if(inst->Internal.CoreInt->TypeID != TpCORE_CORE_TYPE_ID){
//						inst->Error = TRUE;
//						inst->ErrorID = trkPAPER_SH_CONTROL_ERR_INVALID_HANDLE;
//
//						inst->Internal.State = trkPAPER_SH_CONTROL_ERROR;
//					}
//					else{
//						inst->Active = TRUE;
//
//						inst->Internal.State = trkPAPER_SH_CONTROL_INIT;
//					}
//				}
//			}
//			break;
//		case trkPAPER_SH_CONTROL_INIT:
//			//******************************************************************************** Init state
//			if(CheckValidity(&inst->SelectedElem)){	//Checking for the validity of the selected element format
//				inst->Internal.Idx = GetIndex(&inst->SelectedElem);	//Pulling the index from the string
//				if(inst->Internal.CoreInt->Axes[inst->Internal.Idx].Present){ //Verifying that index has a valid access in it
//					inst->ErrorID = trkPAPER_SH_CONTROL_ERR_OK;
//					inst->Valid = TRUE;
//					inst->Internal.CurrentAxis = inst->Internal.CoreInt->Axes[inst->Internal.Idx].Axis;
//
//					inst->Internal.Fbs.ShGetInfo.Axis = &inst->Internal.CurrentAxis;
//					inst->Internal.Fbs.ShGetInfo.Enable = TRUE;
//
//					inst->Internal.State = trkPAPER_SH_CONTROL_IDLE;
//				}
//				else{
//					inst->ErrorID = trkPAPER_SH_CONTROL_WARN_SH_NOT_AVAIL;
//				}
//			}
//			else{
//				inst->ErrorID = trkPAPER_SH_CONTROL_WARN_NO_ELEM_FND;
//			}
//
//			break;
//		case trkPAPER_SH_CONTROL_IDLE:
//			//******************************************************************************** Get Shuttle state
//			//Need to check for if the selected element has changed
//			inst->Internal.LastIdx = inst->Internal.Idx;
//			if(CheckValidity(&inst->SelectedElem)){
//				inst->Internal.Idx = GetIndex(&inst->SelectedElem);
//
//				if(inst->Internal.Idx != inst->Internal.LastIdx){
//					//We've changed indecies need to head back to init to reset the sh status
//					inst->Valid = FALSE;
//					inst->Internal.Fbs.ShGetInfo.Enable = FALSE;
//
//					inst->Internal.State = trkPAPER_SH_CONTROL_INIT;
//				}
//				else{
//					//Here we can start parsing commands
//					if(inst->ElasticMoveAbs){
//						//Setup the elastic move absolute block and execute it
//						inst->Internal.Fbs.ElMoveAbs.Axis = &inst->Internal.CurrentAxis;
//						inst->Internal.Fbs.ElMoveAbs.Position = inst->Parameters->Position;
//						inst->Internal.Fbs.ElMoveAbs.Velocity = inst->Parameters->Vel;
//						inst->Internal.Fbs.ElMoveAbs.Acceleration = inst->Parameters->Accel;
//						inst->Internal.Fbs.ElMoveAbs.Deceleration = inst->Parameters->Decel;
//
//						inst->Internal.Fbs.ElMoveAbs.Execute = TRUE;
//
//						inst->Internal.State = trkPAPER_SH_CONTROL_EL_MOVE_ABS;
//					}
//					else if(inst->ElasticMoveAdd){
//						//Setup the elastic move additve block and execute it
//						inst->Internal.Fbs.ElMoveAdd.Axis = &inst->Internal.CurrentAxis;
//						inst->Internal.Fbs.ElMoveAdd.Distance = inst->Parameters->Distance;
//						inst->Internal.Fbs.ElMoveAdd.Velocity = inst->Parameters->Vel;
//						inst->Internal.Fbs.ElMoveAdd.Acceleration = inst->Parameters->Accel;
//						inst->Internal.Fbs.ElMoveAdd.Deceleration = inst->Parameters->Decel;
//
//						inst->Internal.Fbs.ElMoveAdd.Execute = TRUE;
//
//						inst->Internal.State = trkPAPER_SH_CONTROL_EL_MOVE_ADD;
//					}//End of commands check conditionals
//				}
//			}
//			else{//We've received an invalid selection, need to reset the flags and Sh Status
//				inst->Valid = FALSE;
//				inst->Internal.Fbs.ShGetInfo.Enable = FALSE;
//
//				inst->Internal.State = trkPAPER_SH_CONTROL_INIT;
//			}
//
//			break;
//		case trkPAPER_SH_CONTROL_EL_MOVE_ABS:
//			//******************************************************************************** Elastic Move absolute state
//			if(inst->Internal.Fbs.ElMoveAbs.Error){
//				inst->Error = TRUE;
//				inst->ErrorID = trkPAPER_SH_CONTROL_ERR_EL_MOVE;
//
//				inst->Internal.State = trkPAPER_SH_CONTROL_ERROR;
//			}
//			else if(inst->Internal.Fbs.ElMoveAbs.Active){
//				inst->MovementActive = TRUE;
//				inst->Internal.Fbs.ElMoveAbs.Execute = FALSE;
//
//				inst->Internal.LastIdx = inst->Internal.Idx;
//				if(CheckValidity(&inst->SelectedElem)){
//					inst->Internal.Idx = GetIndex(&inst->SelectedElem);
//
//					if(inst->Internal.Idx != inst->Internal.LastIdx){
//						//We've changed indecies need to head back to init to reset the sh status
//						inst->Valid = FALSE;
//						inst->Internal.Fbs.ShGetInfo.Enable = FALSE;
//
//						inst->Internal.State = trkPAPER_SH_CONTROL_INIT;
//					}
//				}
//			}
//			else if(inst->Internal.Fbs.ElMoveAbs.Done){
//				inst->Internal.Fbs.ElMoveAbs.Execute = FALSE;
//				inst->MovementActive = FALSE;
//				inst->MovementDone = TRUE;
//
//				inst->Internal.State = trkPAPER_SH_CONTROL_MOVE_DONE;
//			}
//			break;
//		case trkPAPER_SH_CONTROL_EL_MOVE_ADD:
//			//******************************************************************************** Elastic Move Additive state
//			if(inst->Internal.Fbs.ElMoveAdd.Error){
//				inst->Error = TRUE;
//				inst->ErrorID = trkPAPER_SH_CONTROL_ERR_EL_MOVE;
//
//				inst->Internal.State = trkPAPER_SH_CONTROL_ERROR;
//			}
//			else if(inst->Internal.Fbs.ElMoveAdd.Done){
//				inst->MovementActive = FALSE;
//				inst->MovementDone = TRUE;
//
//				inst->Internal.Fbs.ElMoveAdd.Execute = FALSE;
//
//				inst->Internal.State = trkPAPER_SH_CONTROL_MOVE_DONE;
//			}
//			else{
//				inst->MovementActive = TRUE;
//			}
//			break;
//		case trkPAPER_SH_CONTROL_MOVE_DONE:
//			//******************************************************************************** Movement Done State
//			if(!inst->ElasticMoveAbs
//				&& !inst->ElasticMoveAdd){
//				inst->MovementDone = FALSE;
//
//				inst->Internal.State = trkPAPER_SH_CONTROL_IDLE;
//			}
//			break;
//		case trkPAPER_SH_CONTROL_ERROR:
//			//******************************************************************************** Error State
//			if(!inst->Enable){
//				inst->Error = FALSE;
//				inst->ErrorID = trkPAPER_SH_CONTROL_ERR_OK;
//
//				inst->Internal.Fbs.ElMoveAbs.Execute = FALSE;
//				inst->Internal.Fbs.ElMoveAdd.Execute = FALSE;
//				inst->Internal.Fbs.ShGetInfo.Enable = FALSE;
//
//				inst->Internal.Idx = 0;
//				inst->Internal.LastIdx = 0;
//
//				inst->Internal.State = trkPAPER_SH_CONTROL_OFF;
//			}
//			break;
//	}
//	//FB calls
//
//	MC_BR_ShReadInfo_AcpTrak(&inst->Internal.Fbs.ShGetInfo);
//	MC_BR_ElasticMoveAbs_AcpTrak(&inst->Internal.Fbs.ElMoveAbs);
//	MC_BR_ElasticMoveAdd_AcpTrak(&inst->Internal.Fbs.ElMoveAdd);
}
```

#### TrkPaperShuttleFeature.c
```c
#include <bur/plctypes.h>
#include <stdint.h>
#include <AsBrStr.h>

#define TRUE 1
#define FALSE 0

#ifdef __cplusplus
	extern "C"
	{
#endif
#include "TrkPaper.h"
#ifdef __cplusplus
	};
#endif

//Function Declaration to remove compiler warnings

//Verify that the two string lengths do not exceed a length
plcbit CheckStrLen(char* dest,char* source,UDINT length);

void TrkPaperShuttleFeature(struct TrkPaperShuttleFeature* inst)
{
	DINT BuildShuttlePolygon(char* dest,
	USINT idx,
	LREAL length,
	LREAL width,
	UDINT userDataAdr,
	struct TrkPaperCoreColorOptionType* colorOption){

		char tmp[150];
		USINT red,blue,green;

		if(!colorOption->Enabled){
			snprintf2(tmp,150,"<polygon id=\"sh%d\" points=\"0,0 %0f,0 , %f,%f %f,%f 0,%f\" style=\"fill:rgb(0,255,0);\"/>",
				idx,	//polygon index
				(length-width/2.0),//p1.x
				length,	//p1.y
				width/2.0, //p2.x
				(length-width/2.0),//p2.y
				width,//p2.x
				width); //p3.y
		}
		else{
			brsmemcpy((uintptr_t)&red,userDataAdr + colorOption->Offsets.Red,sizeof(USINT));
			brsmemcpy((uintptr_t)&green,userDataAdr + colorOption->Offsets.Green,sizeof(USINT));
			brsmemcpy((uintptr_t)&blue,userDataAdr + colorOption->Offsets.Blue,sizeof(USINT));

			snprintf2(tmp,150,"<polygon id=\"sh%d\" points=\"0,0 %0f,0 , %f,%f %f,%f 0,%f\" style=\"fill:rgb(%d,%d,%d);\"/>",
				idx,	//polygon index
				(length-width/2.0),//p1.x
				length,	//p1.y
				width/2.0, //p2.x
				(length-width/2.0),//p2.y
				width,//p2.x
				width,
				red,
				green,
				blue); //p3.y
		}
		if(CheckStrLen(dest,(char*)&tmp,trkPAPER_CORE_MAX_STR_LEN)){
			brsstrcat((uintptr_t)dest,(uintptr_t)&tmp);
			return trkPAPER_CORE_ERR_OK;
		}
		else
			return trkPAPER_CORE_ERR_STR_LEN_EXCD;
	}
	//This function loops through the assembly monitor data and builds a SVG string + SVG Transform. Will return 0 if succesful
	//Will monitor to make sure the string lengths are not exceeded
	DINT BuildShuttleStrings(struct McAcpTrakAssemblyMonData* mon,
	char* svgContent,char* svgTransform,
	struct TrkPaperCoreOptionsType* coreOptions){
		USINT i;
		USINT transCounter;
		transCounter = 0;
		char tmp[150];

		for (i = 0; i < trkPAPER_MAX_SHUTTLE_COUNT; i++){
			if(mon->Shuttle[i].Available){
				brsmemset((uintptr_t)&tmp,0,sizeof(tmp));

				LREAL width;
				LREAL length;
				LREAL shCenterX;
				LREAL shCenterY;

				width = mon->Shuttle[i].Width / 1000.0;
				length = (mon->Shuttle[i].ExtentToBack + mon->Shuttle[i].ExtentToFront)/ 1000.0;
				shCenterX = mon->Shuttle[i].Position.X / 1000.0 - mon->Shuttle[i].ExtentToBack / 1000.0;
				shCenterY = -(mon->Shuttle[i].Position.Y / 1000.0 + width / 2.0);

				snprintf2(tmp,150,"<g id=\"Shuttle%d\">",mon->Shuttle[i].Index);
				if(CheckStrLen(svgContent,(char*)&tmp,trkPAPER_CORE_MAX_STR_LEN)){
					brsstrcat((uintptr_t)svgContent,(uintptr_t)&tmp);
				}
				else
					return trkPAPER_CORE_ERR_STR_LEN_EXCD;

				DINT returnVal;
				returnVal = BuildShuttlePolygon(svgContent,mon->Shuttle[i].Index,length,width,mon->Shuttle[i].UserData,&coreOptions->Color);
				if(returnVal!= trkPAPER_CORE_ERR_OK)
					return returnVal;

				snprintf2(tmp,150,"<text x=\"%f\" y=\"%f\" font-weight=\"bold\" font-size=\"0.035px\">%d</text>",
					mon->Shuttle[i].ExtentToBack / 2000.0,
					width * 3.0 / 4.0,
					mon->Shuttle[i].Index);
				if(CheckStrLen(svgContent,(char*)&tmp,trkPAPER_CORE_MAX_STR_LEN)){
					brsstrcat((uintptr_t)svgContent,(uintptr_t)&tmp);
				}
				else
					return trkPAPER_CORE_ERR_STR_LEN_EXCD;

				//Create an invisible bounding rectangle to handle the click event. "Invisible" by using the alpha channel, if you use the
				//Vibisility property, the click event will not fire for the SVG
				snprintf2(tmp,150,"<rect id=\"ID%d\" width=\"%f\" height=\"%f\" style=\"fill:rgba(0,0,0,0)\"/>",
					mon->Shuttle[i].Index,
					length,
					width);
				if(CheckStrLen(svgContent,(char*)&tmp,trkPAPER_CORE_MAX_STR_LEN)){
					brsstrcat((uintptr_t)svgContent,(uintptr_t)&tmp);
				}
				else
					return trkPAPER_CORE_MAX_STR_LEN;

				if(CheckStrLen(svgContent,(char*)&"</g>",trkPAPER_CORE_MAX_STR_LEN)){
					brsstrcat((uintptr_t)svgContent,(uintptr_t)&"</g>");
				}
				else
					return trkPAPER_CORE_ERR_STR_LEN_EXCD;

				//Check to see if we've had more transforms to add a comma between the units
				if(transCounter>0){
					if(CheckStrLen(svgTransform,(char*)&",",trkPAPER_CORE_MAX_STR_LEN)){
						brsstrcat((uintptr_t)svgTransform,(uintptr_t)&",");
					}
					else
						return trkPAPER_CORE_ERR_STR_LEN_EXCD;
				}
				//Preform translation
				snprintf2(tmp,150,"{\"select\":\"#Shuttle%d\",\"duration\":100,\"display\":true,\"translate\":[%f,%f]},",
					mon->Shuttle[i].Index,
					shCenterX,
					shCenterY,
					-mon->Shuttle[i].Orientation.Angle1,
					length/2.0,
					width/2.0);
				if(CheckStrLen(svgTransform,(char*)&tmp,trkPAPER_CORE_MAX_STR_LEN)){
					brsstrcat((uintptr_t)svgTransform,(uintptr_t)&tmp);
				}
				else
					return trkPAPER_CORE_ERR_STR_LEN_EXCD;
				//Preform rotation
				snprintf2(tmp,150,"{\"select\":\"#sh%d\",\"duration\":100,\"display\":true,\"spin\":[%f,%f,%f]}",
					mon->Shuttle[i].Index,
					-mon->Shuttle[i].Orientation.Angle1, //Spin amount
					length/2.0,	//Spin center x
					width/2.0); //Spin center y
				if(CheckStrLen(svgTransform,(char*)&tmp,trkPAPER_CORE_MAX_STR_LEN)){
					brsstrcat((uintptr_t)svgTransform,(uintptr_t)&tmp);
				}
				else
					return trkPAPER_CORE_ERR_STR_LEN_EXCD;
				transCounter++;
			}

		}

		//No Error, finished everything return OK
		return trkPAPER_CORE_ERR_OK;
	}
}
```

- SvgPrep.py (not shown)

#### README.md
~~~~markdown
# Track Paper Widget Library
This is a brief overview of how to implement the track paper widget.

## Overview
The track paper widget library provides a convenient wrapper to automatically build the SVG strings for an entire track system for the paper widget. The library utilizes the prebuilt SVG from the track system (post processed) in combination with acp trak status blocks to build a simple drop in widget to show the status of an acp trak system.

# Major Components
The TrakPaper widget consists of a few components.
1. TrakPaper Library
2. TrakDiag Task
3. SegmentStatus Custom Widget
4. MpPaper widget
5. ACOPOS Trak layout generated SVG

Each of these components works together to create the TrakMap widget and functionality.

## Usage
### Preparing the SVG
   The first step to use the track map is to have the automatically generated SVG generated with a valid layout and the SVGData file device. Some simple post processing must be done on this SVG in order to function with the Trak Paper widget. The SVG must be generated from a system with MpMotion 5.13+. The post processing is done by executing the SvgPython.py script with the input file name of the pre-generated SVG. To run the script you will need to have Python (preferably 3.8+) installed

   1. Place SvgPrep.py and generated SVG into the same directory
   2. Open a command line in this directory
   3. Type `python SvgPrep.py -i preGeneratedSvg.svg -o OutputFileName.svg`
      1. You can enter the command with or without the file extensions

Upon a success a new file named "OutputFileName.svg" will have been generated in the same directory. This is the new pre-processed SVG that you will use in the paper widget.

### Add in the Track Paper Library
To your project add the track paper library and the "TrakDiag" task. The TrakDiag task is the task that automatically implements the TrakPaper Core function block and supporting function blocks.

### Populate the Segment List Variable
The TrakPaper library uses a list of segments to build the string. In order for this to work you must populate a segment list with the segment variable reference and the name of that segment. The variable is TrackDiag.Seg.SegList.

The easiest method is in your init of the task add your definitions for the segments:

    TrackDiag.Seg.SegList[0].Name  := 'gSeg_A_1'; 	TrackDiag.Seg.SegList[0].McType := gSeg_A_1;
    TrackDiag.Seg.SegCount := 1;

The above would make a system with a singular segment with a segment name of gSeg_A_1.

### Setting up the Paper widget
The final step that must be done is to connect to the paper widget and custom status widget.
#### Paper Widget
To the paper widget, map the paperCore variable SvgTransform and SvgContent variables from the TrakDiag task (you will likely need to enable the two variables via OPC-UA first).

The Trak paper widget uses the color List property of the paper widget for the segment status colors during operation. The default color values could be the following: `#c9c9c9,#FF0000,#00FF00,#FFFF80`
The important is that the following indices are used for the styling of the segments:

| Style Description | Index |
| ------ | ------ |
| Segment Default Style | 0 |
| Segment is in an error state | 1 |
| Segment is okay style | 2 |
| Segment is in a warning state style | 3 |

Custom styling is possible by changing the color at the defined index.

In order to use the segment details, the "clickID" property must be set for the Paper Widget. This can be done by using the below code block in an event binding and setting the "contentRefId" and "widgetRefId" correctly
```xml
<?xml version="1.0" encoding="utf-8"?>
<EventBindingSet id="trackmapContent_eventbinding" xmlns="http://www.br-automation.com/iat2014/eventbinding/v2" xmlns:types="http://www.br-automation.com/iat2015/widgetTypes/v2" xmlns:xsi="http://www.w3.org/2001/XMLSchema-instance">
  <Bindings>
    <EventBinding id="content_trackmap.paperTrackMap.Click">
      <Source xsi:type="widgets.brease.Paper.Event" contentRefId="trackmapContent" widgetRefId="paperTrackMap" event="Click" />
      <EventHandler>
        <Action>
          <Target xsi:type="opcUa.NodeAction" refId="TrackDiag:clickId">
            <Method xsi:type="opcUa.NodeAction.SetValueString" value="= elementId" />
          </Target>
        </Action>
      </EventHandler>
    </EventBinding>
  </Bindings>
</EventBindingSet>
```

#### Custom Status Widget
To use the custom widget, add the custom library provided into the project. Add the SegmentStatus widget into your content wherever you desire. Connect the `TrackDiag:clickedSegment` variable to the widget. That is all that is needed for the custom widget

#### Text Files
In the provided files there are the text files. These can be included to populate the error texts and segment statuses in the status widget. Add the provided text files to the text definition for the project.
~~~~

#### Types.typ - not listed in the package file held
```iecst
(*Track Master Core Types*)

TYPE
	tpCoreInternalTyp : 	STRUCT  (*Internal Datatype*)
		TypeID : UDINT; (*TypeID to help with handle application*)
		State : USINT; (*State of execution*)
	END_STRUCT;
	tpCoreViewBoxCfgTyp : 	STRUCT  (*Attributes of the SVG's viewbox*)
		MinX : REAL; (*Minimum x position*)
		MinY : REAL; (*minimum y position*)
		Width : REAL; (*Width of viewbox*)
		Height : REAL; (*Height of viewbox*)
	END_STRUCT;
	tpCoreStateEnum :
		( (*State of execution*)
		tpCORE_OFF, (*Waiting for enable command*)
		tpCORE_INIT, (*Initialization state*)
		tpCORE_RUNNING, (*Running state*)
		tpCORE_RESET, (*Resetting state*)
		tpCORE_ERROR (*Error state*)
		);
	tpCoreErrorEnum :
		( (*Error Enumeration*)
		tpCORE_ERR_OK := 0, (*No error present*)
		tpCORE_ERR_INVALID_ASSEMBLY := -61000, (*Invalid input assembly reference*)
		tpCORE_ERR_SH_COUNT_EXCEEDED := -61001, (*Maximum shuttle count exceeded. Need to increase max shuttle count constant*)
		tpCORE_ERR_STR_LEN_EXCEEDED := -61002 (*The built string is too long, need to increase the maximum size to prevent page faulting*)
		);
	tpCoreSvgLengthsTyp : 	STRUCT  (*String lengths of SVGs*)
		ContentLength : UDINT; (*String Length of SVG Content string*)
		TransformLength : UDINT; (*String Length of SVG Transform string*)
	END_STRUCT;
	tpCoreAxisLookupTyp : 	STRUCT  (*Lookup table datatype*)
		Present : BOOL; (*Axis is present and a valid reference exists*)
		Axis : McAxisType; (*Axis information*)
	END_STRUCT;
	tpCoreOptionsTyp : 	STRUCT  (*Options for Core Function Block*)
		Color : tpCoreColorOptionTyp; (*Shuttle Color Option*)
		Shuttle : tpCoreShuttleOptionTyp; (*Shuttle Option*)
	END_STRUCT;
	tpCoreShuttleOptionTyp : 	STRUCT  (*Shuttle Option*)
		Enabled : BOOL; (*Option is enabled*)
	END_STRUCT;
	tpSegmentStyleEnumeration :
		( (*Style enumeration for the track map strings*)
		segStyleDefault := 0, (*Segment Default Style*)
		segStyleError := 1, (*Segment is in error style*)
		segStyleOkay := 2, (*Segment is okay style*)
		segStyleWarning := 3 (*Segment is in a warning state style*)
		);
	tpCoreColorOptionTyp : 	STRUCT  (*Shuttle Color Option*)
		Enabled : BOOL; (*Option is enabled*)
		Offsets : tpCoreColorOffsetsTyp; (*Userdata color offsets*)
	END_STRUCT;
	tpCoreColorOffsetsTyp : 	STRUCT  (*Userdata color offsets*)
		Red : UDINT; (*Offset for UserData address for the Red color in USINT*)
		Green : UDINT; (*Offset for UserData address for the Green color in USINT*)
		Blue : UDINT; (*Offset for UserData address for the Blue color in USINT*)
	END_STRUCT;
	tpCoreSegmentTyp : 	STRUCT
		Name : STRING[32]; (*Name of the segment in the SVG*)
		McType : McSegmentType; (*Segment Reference*)
		Status : tpCoreSegmentStatusTyp; (*Status Information for the segment*)
	END_STRUCT;
	tpCoreSegmentStatusTyp : 	STRUCT
		CommunicationReady : BOOL; (*Communication ready on the segment*)
		ReadyForPowerOn : BOOL; (*Segment is ready for power on*)
		PowerOn : BOOL; (*Segment is powered*)
		StartupCount : UDINT; (*Number of startups on the segment*)
		CommunicationState : McCommunicationStateEnum; (*Communication state of the segment*)
		SegmentDisabled : BOOL; (*Segment is disabled*)
		SegmentReady : BOOL; (*Segment is Ready*)
		SegmentStopping : BOOL; (*Segment is in the Stopping State*)
		SegmentErrorStop : BOOL; (*Segment is in an error stop state*)
		ErrorCode : UINT; (*Error code of the segment*)
		DCBus : SegStatusDCBus_typ;
		Temp : SegStatusTemp_typ;
	END_STRUCT;
END_TYPE

(*Track Master Shuttle Control Types*)

TYPE
	tpShuttleControlParsTyp : 	STRUCT  (*Input parameters for Shuttle Control*)
		Position : LREAL; (*Destination position for Absolute and Velocity commands*)
		Distance : LREAL; (*Distance for all relative commands*)
		Vel : REAL; (*Comanded Movement velocity*)
		Accel : REAL; (*Comanded Movement acceleration*)
		Decel : REAL; (*Comanded Movement deceleration*)
	END_STRUCT;
	tpShuttleControlInternalTyp : 	STRUCT  (*Internal data type*)
		State : tpShuttleControlStatesEnum; (*State of execution*)
		CoreInt : REFERENCE TO tpCoreInternalTyp; (*Internal data for the Core function block*)
		CurrentAxis : McAxisType; (*Current selected Axis*)
		Fbs : tpShuttleControlFbTyp; (*Internal function blocks*)
		Idx : USINT; (*Selected Index for the axis lookup table*)
		LastIdx : USINT; (*Last cycle selected index for the axis lookup table*)
	END_STRUCT;
	tpShuttleControlFbTyp : 	STRUCT  (*Internal Function Blocks*)
		ShGetInfo : MC_BR_ShReadInfo_AcpTrak; (*Shuttle Get info*)
		ElMoveAbs : MC_BR_ElasticMoveAbs_AcpTrak; (*Elastic move absolute command*)
		ElMoveAdd : MC_BR_ElasticMoveAdd_AcpTrak; (*Elastic move addtive command*)
	END_STRUCT;
	tpShuttleControlErrorEnum :
		( (*Error enumeration*)
		tpSH_CONTROL_ERR_OK := 0, (*No error currently*)
		tpSH_CONTROL_WARN_SH_NOT_AVAIL := -52000, (*Shuttle Currently not listed as available*)
		tpSH_CONTROL_WARN_NO_ELEM_FND := -52001, (*Input selected element did not return a shuttle*)
		tpSH_CONTROL_ERR_INVALID_HANDLE := -62000, (*Invalid input handle*)
		tpSH_CONTROL_ERR_EL_MOVE := -62001 (*Error in an elastic movment*)
		);
	tpShuttleControlStatesEnum :
		( (*State of execution*)
		tpSH_CONTROL_OFF, (*Off State*)
		tpSH_CONTROL_INIT, (*Init/Waiting for valid ShElement state*)
		tpSH_CONTROL_IDLE, (*Idle waiting for a command state*)
		tpSH_CONTROL_EL_MOVE_ABS, (*Move Elastic absoulte active state*)
		tpSH_CONTROL_EL_MOVE_ADD, (*Move Elastic Additive active state*)
		tpSH_CONTROL_MOVE_DONE, (*Move has completed*)
		tpSH_CONTROL_ERROR (*Error present on the FB*)
		);
END_TYPE

(*Temporary Segment information*)

TYPE
	SegStatusTemp_typ : 	STRUCT
		TemperatureCON : REAL; (*monitor temperature CON*)
		TemperaturePROZ : REAL; (*monitor temperature PROZ*)
		TemperatureAIR : REAL; (*monitor temperature AIR*)
		TemperatureBAL : REAL; (*monitor temperature BAL*)
		TemperatureCHASSIS_1 : REAL; (*monitor temperature CHASSIS_1*)
		TemperatureCHASSIS_2 : REAL; (*monitor temperature CHASSIS_2*)
		TemperatureCHASSIS_3 : REAL; (*monitor temperature CHASSIS_3*)
		TemperaturePOWER_SENS3 : REAL; (*monitor temperature POWER_SENS3*)
		TemperaturePOWER_SENS4 : REAL; (*monitor temperature POWER_SENS4*)
		TemperaturePOWER_SENS5 : REAL; (*monitor temperature POWER_SENS5*)
		TemperaturePOWER_SENS6 : REAL; (*monitor temperature POWER_SENS6*)
		TemperaturePOWER_SENS7 : REAL; (*monitor temperature POWER_SENS7*)
		TemperaturePOWER_SENS8 : REAL; (*monitor temperature POWER_SENS8*)
		TemperaturePOWER_SENS9 : REAL; (*monitor temperature POWER_SENS9*)
		TemperaturePOWER_SENS10 : REAL; (*monitor temperature POWER_SENS10*)
		TemperaturePOWER_SENS11 : REAL; (*monitor temperature POWER_SENS11*)
	END_STRUCT;
	SegStatusDCBus_typ : 	STRUCT
		DCBusVoltage : REAL;
		DCBusVoltageMax : REAL;
		DCBusVoltageMin : REAL;
	END_STRUCT;
END_TYPE
```

#### Constants.var - not listed in the package file held
```iecst
VAR CONSTANT
	tpMAX_SHUTTLE_COUNT : USINT := 150;
	tpMAX_SHUTLE_ARRAY : USINT := tpMAX_SHUTTLE_COUNT-1;
	tpCORE_CORE_TYPE_ID : DINT := 651684313;
	tpCORE_MAX_STR_LEN : UDINT := 10000;
END_VAR
```

#### tpCore.c - not listed in the package file held
```c
#include <bur/plctypes.h>

#define TRUE 1
#define FALSE 0

#ifdef __cplusplus
	extern "C"
	{
#endif
#include "TrkPaper.h"
#ifdef __cplusplus
	};
#endif
//Verify that the two string lengths do not exceed a length
plcbit CheckStrLen(char* dest,char* source,UDINT length){
	if(brdkStrLen(dest) + brdkStrLen(source) >= length){
		return FALSE;
	}
	else{
		return TRUE;
	}
}

DINT StartSVGStrings(char* svgContent,
	char* svgTransform,
struct tpCoreViewBoxCfgTyp* viewBox){

	char tmp[150];

	brsmemset(svgContent,0,sizeof(svgContent));
	brsmemset(svgTransform,0,sizeof(svgTransform));

	snprintf2(tmp,150,"<svg viewBox=\"%f %f %f %f\">",
		viewBox->MinX,
		viewBox->MinY,
		viewBox->Width,
		viewBox->Height);
	if(CheckStrLen(svgContent,&tmp,tpCORE_MAX_STR_LEN)){
		brsstrcat(svgContent,&tmp);
	}
	else
		return tpCORE_ERR_STR_LEN_EXCEEDED;
	if(CheckStrLen(svgTransform,&"[",tpCORE_MAX_STR_LEN)){
		brsstrcat(svgTransform,&"[");
	}
	else
		return tpCORE_ERR_STR_LEN_EXCEEDED;
	//No Error, finished everything return OK
	return tpCORE_ERR_OK;

}

//Closes the Transform and Content strings with the appropriate tags
DINT CloseSVGStrings(char* svgContent,
char* svgTransform){
	if(CheckStrLen(svgContent,&"</svg>",tpCORE_MAX_STR_LEN)){
		brsstrcat(svgContent,&"</svg>");
	}
	else
		return tpCORE_ERR_STR_LEN_EXCEEDED;
	if(CheckStrLen(svgTransform,&"]",tpCORE_MAX_STR_LEN)){
		brsstrcat(svgTransform,&"]");
	}
	else
		return tpCORE_ERR_STR_LEN_EXCEEDED;

	//No Error, finished everything return OK
	return tpCORE_ERR_OK;
}

//Method for building the shuttle transform string. Defined the style of a segment based upon the information input into the FB
DINT BuildSegmentStrings(char* svgContent,
	char* svgTransform,
struct tpCoreSegmentTyp* segList,
USINT SegmentCount){

	USINT i;
	char tmp[200];

	//{"select":"#Segment","fill":1"}
	for (i = 0; i < SegmentCount; i++){
		if(segList[i].Status.ErrorCode > 0){
			snprintf2(tmp,200,"{\"select\":\"#%s\",\"style\":\"fill:%d\"}",
				segList[i].Name, //Segment Name
				segStyleError //Segment Style Color index
				);

		}
		else if(!segList[i].Status.CommunicationReady || !segList[i].Status.ReadyForPowerOn){
			snprintf2(tmp,200,"{\"select\":\"#%s\",\"style\":\"fill:%d\"}",
				segList[i].Name, //Segment Name
				segStyleWarning //Segment Style Color index
				);
		}
		else if(segList[i].Status.PowerOn){
			snprintf2(tmp,200,"{\"select\":\"#%s\",\"style\":\"fill:%d\"}",
				segList[i].Name, //Segment Name
				segStyleOkay //Segment Style Color index
				);
		}
		else{
			snprintf2(tmp,200,"{\"select\":\"#%s\",\"style\":\"fill:%d\"}",
				segList[i].Name, //Segment Name
				segStyleDefault //Segment Style Color index
				);
		}

		if(CheckStrLen(svgTransform,&tmp,tpCORE_MAX_STR_LEN)){
			brsstrcat(svgTransform,&tmp);
			if(CheckStrLen(svgTransform,&",",tpCORE_MAX_STR_LEN)){
				//Every one except for the last index add a comma
				if(i != SegmentCount-1){
					brsstrcat(svgTransform,&",");
				}
			}
			else{
				return tpCORE_ERR_STR_LEN_EXCEEDED;
			}

		}
		else
			return tpCORE_ERR_STR_LEN_EXCEEDED;
	}

	return tpCORE_ERR_OK;

}

/* Core Track Master function blocks. Handles the building of the SVG string */
void tpCore(struct tpCore* inst)
{
	switch (inst->Internal.State){
		case tpCORE_OFF:
			//******************************************************************************** Off state
			if(inst->Enable){
				inst->Internal.TypeID = tpCORE_CORE_TYPE_ID;
				inst->Handle = &inst->Internal;

				inst->Active = TRUE;
				inst->Internal.State = tpCORE_INIT;
			}
			break;
		case tpCORE_INIT:
				inst->Internal.State = tpCORE_RUNNING;
			break;

		case tpCORE_RUNNING:
			StartSVGStrings(&inst->SvgContent,&inst->SvgTransform,&inst->ViewBoxCfg);

			inst->ErrorID = BuildSegmentStrings(&inst->SvgContent,&inst->SvgTransform,inst->Segments,inst->SegmentCount);

			CloseSVGStrings(&inst->SvgContent,&inst->SvgTransform);
			inst->StrLengths.ContentLength = brdkStrLen(&inst->SvgContent);
			inst->StrLengths.TransformLength = brdkStrLen(&inst->SvgTransform);

			if(inst->ErrorID != tpCORE_ERR_OK){
				inst->Error = TRUE;

				inst->Internal.State = tpCORE_ERROR;
			}
			if(!inst->Enable){
				inst->Active = FALSE;
				inst->Internal.State = tpCORE_OFF;
			}
			break;
		case tpCORE_RESET:
			//Try and recover by resetting any blocks

			break;
		case tpCORE_ERROR:
			if(inst->ErrorRest){
				inst->Error = FALSE;
				inst->ErrorID = tpCORE_ERR_OK;

				inst->Internal.State = tpCORE_OFF;
			}
			break;
	}
	//FB calls
}
```

#### tpShuttleControl.c - not listed in the package file held
```c
#include <bur/plctypes.h>

#define TRUE 1
#define FALSE 0

#ifdef __cplusplus
	extern "C"
	{
#endif
#include "TrkPaper.h"
#ifdef __cplusplus
	};
#endif

plcbit CheckValidity(char* selectedElem){
	char buf[2];
	//Get a substring of the first 3 characters
	brdkStrSubStr(&buf,selectedElem,0,3);
	//Look at the start of the selectedID, if it starts with #ID then we know a shuttle has been clicked
	if(0 == brsstrcmp(&buf,&"#ID")){
		return TRUE;
	}
	else{
		return FALSE;
	}
}
USINT GetIndex(char* selectedElem){
	char buf[3];
	brdkStrSubStr(&buf,selectedElem,3,brdkStrLen(selectedElem) - 3);
	return (USINT)brdkStrAToUdint(&buf,BRDK_STR_CONVERT_DECIMAL);
}
/* Function block for handling a shuttle control provided from the paper element's selected element ID. Must be paired with the tmCore FB */
void tpShuttleControl(struct tpShuttleControl* inst)
{
	if(inst->Valid){
		inst->ShInfo = inst->Internal.Fbs.ShGetInfo.ShuttleInfo;
	}
	switch (inst->Internal.State){
		case tpSH_CONTROL_OFF:
			//******************************************************************************** Off state
			if(inst->Enable){
				if(inst->Handle == 0){
					inst->Error = TRUE;
					inst->ErrorID = tpSH_CONTROL_ERR_INVALID_HANDLE;

					inst->Internal.State = tpSH_CONTROL_ERROR;
				}
				else{
					inst->Internal.CoreInt = (tpCoreInternalTyp*)inst->Handle;
					if(inst->Internal.CoreInt->TypeID != tpCORE_CORE_TYPE_ID){
						inst->Error = TRUE;
						inst->ErrorID = tpSH_CONTROL_ERR_INVALID_HANDLE;

						inst->Internal.State = tpSH_CONTROL_ERROR;
					}
					else{
						inst->Active = TRUE;

						inst->Internal.State = tpSH_CONTROL_INIT;
					}
				}
			}
			break;
		case tpSH_CONTROL_INIT:
			//******************************************************************************** Init state
			if(CheckValidity(&inst->SelectedElem)){	//Checking for the validity of the selected element format
				inst->Internal.Idx = GetIndex(&inst->SelectedElem);	//Pulling the index from the string
				if(inst->Internal.CoreInt->Axes[inst->Internal.Idx].Present){ //Verifying that index has a valid access in it
					inst->ErrorID = tpSH_CONTROL_ERR_OK;
					inst->Valid = TRUE;
					inst->Internal.CurrentAxis = inst->Internal.CoreInt->Axes[inst->Internal.Idx].Axis;

					inst->Internal.Fbs.ShGetInfo.Axis = &inst->Internal.CurrentAxis;
					inst->Internal.Fbs.ShGetInfo.Enable = TRUE;

					inst->Internal.State = tpSH_CONTROL_IDLE;
				}
				else{
					inst->ErrorID = tpSH_CONTROL_WARN_SH_NOT_AVAIL;
				}
			}
			else{
				inst->ErrorID = tpSH_CONTROL_WARN_NO_ELEM_FND;
			}

			break;
		case tpSH_CONTROL_IDLE:
			//******************************************************************************** Get Shuttle state
			//Need to check for if the selected element has changed
			inst->Internal.LastIdx = inst->Internal.Idx;
			if(CheckValidity(&inst->SelectedElem)){
				inst->Internal.Idx = GetIndex(&inst->SelectedElem);

				if(inst->Internal.Idx != inst->Internal.LastIdx){
					//We've changed indecies need to head back to init to reset the sh status
					inst->Valid = FALSE;
					inst->Internal.Fbs.ShGetInfo.Enable = FALSE;

					inst->Internal.State = tpSH_CONTROL_INIT;
				}
				else{
					//Here we can start parsing commands
					if(inst->ElasticMoveAbs){
						//Setup the elastic move absolute block and execute it
						inst->Internal.Fbs.ElMoveAbs.Axis = &inst->Internal.CurrentAxis;
						inst->Internal.Fbs.ElMoveAbs.Position = inst->Parameters->Position;
						inst->Internal.Fbs.ElMoveAbs.Velocity = inst->Parameters->Vel;
						inst->Internal.Fbs.ElMoveAbs.Acceleration = inst->Parameters->Accel;
						inst->Internal.Fbs.ElMoveAbs.Deceleration = inst->Parameters->Decel;

						inst->Internal.Fbs.ElMoveAbs.Execute = TRUE;

						inst->Internal.State = tpSH_CONTROL_EL_MOVE_ABS;
					}
					else if(inst->ElasticMoveAdd){
						//Setup the elastic move additve block and execute it
						inst->Internal.Fbs.ElMoveAdd.Axis = &inst->Internal.CurrentAxis;
						inst->Internal.Fbs.ElMoveAdd.Distance = inst->Parameters->Distance;
						inst->Internal.Fbs.ElMoveAdd.Velocity = inst->Parameters->Vel;
						inst->Internal.Fbs.ElMoveAdd.Acceleration = inst->Parameters->Accel;
						inst->Internal.Fbs.ElMoveAdd.Deceleration = inst->Parameters->Decel;

						inst->Internal.Fbs.ElMoveAdd.Execute = TRUE;

						inst->Internal.State = tpSH_CONTROL_EL_MOVE_ADD;
					}//End of commands check conditionals
				}
			}
			else{//We've received an invalid selection, need to reset the flags and Sh Status
				inst->Valid = FALSE;
				inst->Internal.Fbs.ShGetInfo.Enable = FALSE;

				inst->Internal.State = tpSH_CONTROL_INIT;
			}

			break;
		case tpSH_CONTROL_EL_MOVE_ABS:
			//******************************************************************************** Elastic Move absolute state
			if(inst->Internal.Fbs.ElMoveAbs.Error){
				inst->Error = TRUE;
				inst->ErrorID = tpSH_CONTROL_ERR_EL_MOVE;

				inst->Internal.State = tpSH_CONTROL_ERROR;
			}
			else if(inst->Internal.Fbs.ElMoveAbs.Active){
				inst->MovementActive = TRUE;
				inst->Internal.Fbs.ElMoveAbs.Execute = FALSE;

				inst->Internal.LastIdx = inst->Internal.Idx;
				if(CheckValidity(&inst->SelectedElem)){
					inst->Internal.Idx = GetIndex(&inst->SelectedElem);

					if(inst->Internal.Idx != inst->Internal.LastIdx){
						//We've changed indecies need to head back to init to reset the sh status
						inst->Valid = FALSE;
						inst->Internal.Fbs.ShGetInfo.Enable = FALSE;

						inst->Internal.State = tpSH_CONTROL_INIT;
					}
				}
			}
			else if(inst->Internal.Fbs.ElMoveAbs.Done){
				inst->Internal.Fbs.ElMoveAbs.Execute = FALSE;
				inst->MovementActive = FALSE;
				inst->MovementDone = TRUE;

				inst->Internal.State = tpSH_CONTROL_MOVE_DONE;
			}
			break;
		case tpSH_CONTROL_EL_MOVE_ADD:
			//******************************************************************************** Elastic Move Additive state
			if(inst->Internal.Fbs.ElMoveAdd.Error){
				inst->Error = TRUE;
				inst->ErrorID = tpSH_CONTROL_ERR_EL_MOVE;

				inst->Internal.State = tpSH_CONTROL_ERROR;
			}
			else if(inst->Internal.Fbs.ElMoveAdd.Done){
				inst->MovementActive = FALSE;
				inst->MovementDone = TRUE;

				inst->Internal.Fbs.ElMoveAdd.Execute = FALSE;

				inst->Internal.State = tpSH_CONTROL_MOVE_DONE;
			}
			else{
				inst->MovementActive = TRUE;
			}
			break;
		case tpSH_CONTROL_MOVE_DONE:
			//******************************************************************************** Movement Done State
			if(!inst->ElasticMoveAbs
				&& !inst->ElasticMoveAdd){
				inst->MovementDone = FALSE;

				inst->Internal.State = tpSH_CONTROL_IDLE;
			}
			break;
		case tpSH_CONTROL_ERROR:
			//******************************************************************************** Error State
			if(!inst->Enable){
				inst->Error = FALSE;
				inst->ErrorID = tpSH_CONTROL_ERR_OK;

				inst->Internal.Fbs.ElMoveAbs.Execute = FALSE;
				inst->Internal.Fbs.ElMoveAdd.Execute = FALSE;
				inst->Internal.Fbs.ShGetInfo.Enable = FALSE;

				inst->Internal.Idx = 0;
				inst->Internal.LastIdx = 0;

				inst->Internal.State = tpSH_CONTROL_OFF;
			}
			break;
	}
	//FB calls

	MC_BR_ShReadInfo_AcpTrak(&inst->Internal.Fbs.ShGetInfo);
	MC_BR_ElasticMoveAbs_AcpTrak(&inst->Internal.Fbs.ElMoveAbs);
	MC_BR_ElasticMoveAdd_AcpTrak(&inst->Internal.Fbs.ElMoveAdd);
}
```

#### tpShuttleFeature.c - not listed in the package file held
```c
#include <bur/plctypes.h>

#define TRUE 1
#define FALSE 0

#ifdef __cplusplus
	extern "C"
	{
#endif
#include "TrkPaper.h"
#ifdef __cplusplus
	};
#endif
void tpShuttleFeature(struct tpShuttleFeature* inst)
{
	DINT BuildShuttlePolygon(char* dest,
	USINT idx,
	LREAL length,
	LREAL width,
	UDINT userDataAdr,
	struct tpCoreColorOptionTyp* colorOption){

		char tmp[150];
		USINT red,blue,green;
		struct UserDataTyp* tst;

		if(!colorOption->Enabled){
			snprintf2(tmp,150,"<polygon id=\"sh%d\" points=\"0,0 %0f,0 , %f,%f %f,%f 0,%f\" style=\"fill:rgb(0,255,0);\"/>",
				idx,	//polygon index
				(length-width/2.0),//p1.x
				length,	//p1.y
				width/2.0, //p2.x
				(length-width/2.0),//p2.y
				width,//p2.x
				width); //p3.y
		}
		else{
			brsmemcpy(&red,userDataAdr + colorOption->Offsets.Red,sizeof(USINT));
			brsmemcpy(&green,userDataAdr + colorOption->Offsets.Green,sizeof(USINT));
			brsmemcpy(&blue,userDataAdr + colorOption->Offsets.Blue,sizeof(USINT));

			snprintf2(tmp,150,"<polygon id=\"sh%d\" points=\"0,0 %0f,0 , %f,%f %f,%f 0,%f\" style=\"fill:rgb(%d,%d,%d);\"/>",
				idx,	//polygon index
				(length-width/2.0),//p1.x
				length,	//p1.y
				width/2.0, //p2.x
				(length-width/2.0),//p2.y
				width,//p2.x
				width,
				red,
				green,
				blue); //p3.y
		}
		if(CheckStrLen(dest,&tmp,tpCORE_MAX_STR_LEN)){
			brsstrcat(dest,&tmp);
			return tpCORE_ERR_OK;
		}
		else
			return tpCORE_ERR_STR_LEN_EXCEEDED;
	}
	//This function loops through the assembly monitor data and builds a SVG string + SVG Transform. Will return 0 if succesful
	//Will monitor to make sure the string lengths are not exceeded
	DINT BuildShuttleStrings(struct McAcpTrakAssemblyMonData* mon,
	char* svgContent,char* svgTransform,
	struct tpCoreOptionsTyp* coreOptions){
		USINT i;
		USINT transCounter;
		transCounter = 0;
		char tmp[150];

		for (i = 0; i < tpMAX_SHUTTLE_COUNT; i++){
			if(mon->Shuttle[i].Available){
				brsmemset(&tmp,0,sizeof(tmp));

				LREAL width;
				LREAL length;
				LREAL shCenterX;
				LREAL shCenterY;

				width = mon->Shuttle[i].Width / 1000.0;
				length = (mon->Shuttle[i].ExtentToBack + mon->Shuttle[i].ExtentToFront)/ 1000.0;
				shCenterX = mon->Shuttle[i].Position.X / 1000.0 - mon->Shuttle[i].ExtentToBack / 1000.0;
				shCenterY = -(mon->Shuttle[i].Position.Y / 1000.0 + width / 2.0);

				snprintf2(tmp,150,"<g id=\"Shuttle%d\">",mon->Shuttle[i].Index);
				if(CheckStrLen(svgContent,&tmp,tpCORE_MAX_STR_LEN)){
					brsstrcat(svgContent,&tmp);
				}
				else
					return tpCORE_ERR_STR_LEN_EXCEEDED;

				DINT returnVal;
				returnVal = BuildShuttlePolygon(svgContent,mon->Shuttle[i].Index,length,width,mon->Shuttle[i].UserData,&coreOptions->Color);
				if(returnVal!= tpCORE_ERR_OK)
					return returnVal;

				snprintf2(tmp,150,"<text x=\"%f\" y=\"%f\" font-weight=\"bold\" font-size=\"0.035px\">%d</text>",
					mon->Shuttle[i].ExtentToBack / 2000.0,
					width * 3.0 / 4.0,
					mon->Shuttle[i].Index);
				if(CheckStrLen(svgContent,&tmp,tpCORE_MAX_STR_LEN)){
					brsstrcat(svgContent,&tmp);
				}
				else
					return tpCORE_ERR_STR_LEN_EXCEEDED;

				//Create an invisible bounding rectangle to handle the click event. "Invisible" by using the alpha channel, if you use the
				//Vibisility property, the click event will not fire for the SVG
				snprintf2(tmp,150,"<rect id=\"ID%d\" width=\"%f\" height=\"%f\" style=\"fill:rgba(0,0,0,0)\"/>",
					mon->Shuttle[i].Index,
					length,
					width);
				if(CheckStrLen(svgContent,&tmp,tpCORE_MAX_STR_LEN)){
					brsstrcat(svgContent,&tmp);
				}
				else
					return tpCORE_ERR_STR_LEN_EXCEEDED;

				if(CheckStrLen(svgContent,&"</g>",tpCORE_MAX_STR_LEN)){
					brsstrcat(svgContent,&"</g>");
				}
				else
					return tpCORE_ERR_STR_LEN_EXCEEDED;

				//Check to see if we've had more transforms to add a comma between the units
				if(transCounter>0){
					if(CheckStrLen(svgTransform,&",",tpCORE_MAX_STR_LEN)){
						brsstrcat(svgTransform,&",");
					}
					else
						return tpCORE_ERR_STR_LEN_EXCEEDED;
				}
				//Preform translation
				snprintf2(tmp,150,"{\"select\":\"#Shuttle%d\",\"duration\":100,\"display\":true,\"translate\":[%f,%f]},",
					mon->Shuttle[i].Index,
					shCenterX,
					shCenterY,
					-mon->Shuttle[i].Orientation.Angle1,
					length/2.0,
					width/2.0);
				if(CheckStrLen(svgTransform,&tmp,tpCORE_MAX_STR_LEN)){
					brsstrcat(svgTransform,&tmp);
				}
				else
					return tpCORE_ERR_STR_LEN_EXCEEDED;
				//Preform rotation
				snprintf2(tmp,150,"{\"select\":\"#sh%d\",\"duration\":100,\"display\":true,\"spin\":[%f,%f,%f]}",
					mon->Shuttle[i].Index,
					-mon->Shuttle[i].Orientation.Angle1, //Spin amount
					length/2.0,	//Spin center x
					width/2.0); //Spin center y
				if(CheckStrLen(svgTransform,&tmp,tpCORE_MAX_STR_LEN)){
					brsstrcat(svgTransform,&tmp);
				}
				else
					return tpCORE_ERR_STR_LEN_EXCEEDED;
				transCounter++;
			}

		}

		//No Error, finished everything return OK
		return tpCORE_ERR_OK;
	}
}
```

#### TrkPaperSegClickInfo.c - not listed in the package file held
```c
#include <bur/plctypes.h>
#include <stdint.h>
#include <AsBrStr.h>

#define TRUE 1
#define FALSE 0

#ifdef __cplusplus
	extern "C"
	{
#endif
#include "TrkPaper.h"
#ifdef __cplusplus
	};
#endif

DINT SegmentLookup(	struct TrkDiagSegmentType* segList,
	USINT SegmentCount,
	char* SegmentID,
	TrkDiagSegmentType* Data){

	USINT i;

	for (i = 0; i < SegmentCount; i++){
		if (brsmemcmp(segList[i].Name, SegmentID, 32) == 0){
			brsmemcpy(Data, &segList[i], sizeof(segList[i]));
			return trkPAPER_SEG_INFO_ERR_OK;
		}
	}

	return trkPAPER_SEG_INFO_ERR_BAD_IDENT;
}

void TrkPaperSegClickInfo(struct TrkPaperSegClickInfo* inst)
{
	switch (inst->Internal.State){
		case trkPAPER_SEG_CLICK_INFO_OFF:
			//******************************************************************************** Off state
			if(inst->Enable){
				if(inst->Handle == 0){
					inst->Error = TRUE;
					inst->ErrorID = trkPAPER_SEG_INFO_ERR_INVLID_HDL;

					inst->Internal.State = trkPAPER_SEG_CLICK_INFO_ERROR;
				}
				else{
					inst->Internal.CoreInt = (TrkPaperCoreInternalType*)inst->Handle;
					if(inst->Internal.CoreInt->TypeID != trkPAPER_CORE_CORE_TYPE_ID){
						inst->Error = TRUE;
						inst->ErrorID = trkPAPER_SEG_INFO_ERR_INVLID_HDL;

						inst->Internal.State = trkPAPER_SEG_CLICK_INFO_ERROR;
					}
					else{
						inst->Active = TRUE;

						inst->Internal.State = trkPAPER_SEG_CLICK_INFO_WAIT;

						inst->Internal.SegmentCount = inst->Internal.CoreInt->TrakStatus->Seg.SegCount;
						inst->Internal.SegList = inst->Internal.CoreInt->TrakStatus->Seg.SegList;
					}
				}
			}
			break;

		case trkPAPER_SEG_CLICK_INFO_WAIT:

			if(!inst->Enable){
				inst->Active = FALSE;
				inst->Internal.State = trkPAPER_SEG_CLICK_INFO_OFF;
			}else if(inst->Update){
				inst->Valid = FALSE;
				inst->Internal.State = trkPAPER_SEG_CLICK_INFO_LOOKUP;
			}

			break;

		case trkPAPER_SEG_CLICK_INFO_LOOKUP:
			inst->ErrorID = SegmentLookup(inst->Internal.SegList, inst->Internal.SegmentCount, (char*)&inst->Ident, &inst->Data);

			if(inst->ErrorID != trkPAPER_SEG_INFO_ERR_OK){
				inst->Error = TRUE;

				inst->Internal.State = trkPAPER_SEG_CLICK_INFO_ERROR;
			}
			else{
				inst->Valid = TRUE;
				inst->Internal.State = trkPAPER_SEG_CLICK_INFO_WAIT;

			}
			break;

		case trkPAPER_SEG_CLICK_INFO_ERROR:
			if(inst->ErrorReset){
				inst->Error = FALSE;
				inst->ErrorID = trkPAPER_SEG_INFO_ERR_OK;

				inst->Internal.State = trkPAPER_SEG_CLICK_INFO_OFF;
			}
			break;
	}
}
```

#### TrkPaperShuttleClickInfo.c - not listed in the package file held
```c
#include <bur/plctypes.h>
#include <stdint.h>
#include <AsBrStr.h>

#define TRUE 1
#define FALSE 0

#ifdef __cplusplus
	extern "C"
	{
#endif
#include "TrkPaper.h"
#ifdef __cplusplus
	};
#endif

DINT ShuttleLookup(struct TrkPaperCoreAxisLookupType* Axes,
	char* ShuttleID,
	TrkPaperShClickInfoDataType* Data,
struct MC_BR_ShReadInfo_AcpTrak* ShReadInfo){

	USINT ShuttleIndex;
	USINT i;

	ShuttleIndex = atoi((uintptr_t)ShuttleID);

	for (i = 0; i < trkPAPER_MAX_SHUTTLE_COUNT; i++){
		if (Axes[i].ShuttleID == ShuttleIndex){
			ShReadInfo->Axis =(uintptr_t)&Axes[i].Axis;
			return FALSE;
		}

		}	return TRUE;
}

void TrkPaperShuttleClickInfo(struct TrkPaperShuttleClickInfo* inst)
{
	switch (inst->Internal.State){
		case trkPAPER_SH_CLICK_INFO_OFF:
			//******************************************************************************** Off state
			if(inst->Enable){
				if(inst->Handle == 0){
					inst->Error = TRUE;
					inst->ErrorID = trkPAPER_SH_INFO_ERR_INVLID_HDL;

					inst->Internal.State = trkPAPER_SH_CLICK_INFO_ERROR;
				}
				else{
					inst->Internal.CoreInt = (TrkPaperCoreInternalType*)inst->Handle;
					if(inst->Internal.CoreInt->TypeID != trkPAPER_CORE_CORE_TYPE_ID){
						inst->Error = TRUE;
						inst->ErrorID = trkPAPER_SH_INFO_ERR_INVLID_HDL;

						inst->Internal.State = trkPAPER_SH_CLICK_INFO_ERROR;
					}
					else{
						inst->Active = TRUE;
						inst->Internal.Fbs.AsmGetShuttle.Assembly = inst->Internal.CoreInt->Assembly;
						inst->Internal.State = trkPAPER_SH_CLICK_INFO_WAIT;
					}
				}
			}
			break;

		case trkPAPER_SH_CLICK_INFO_WAIT:

			//If build table case (power on, shuttle count change) build table
			inst->Valid = FALSE;
			if(inst->Internal.CoreInt->TrakStatus->Asm.PowerOn && inst->Internal.CoreInt->TrakStatus->Asm.AssemblyReady){
				inst->Internal.State = trkPAPER_SH_BUILD_TABLE;
			}
			break;

		case trkPAPER_SH_CLICK_INFO_RUN:

			//Cyclicly read shuttle data
			if(!inst->Internal.CoreInt->TrakStatus->Asm.PowerOn){
				inst->Internal.State = trkPAPER_SH_CLICK_INFO_WAIT;
				inst->Internal.Fbs.ShReadInfo.Enable = FALSE;
				inst->Valid = FALSE;
			}
			else if(!inst->Enable){
				inst->Active = FALSE;
				inst->Valid = FALSE;
				inst->Internal.State = trkPAPER_CORE_OFF;
				inst->Internal.Fbs.ShReadInfo.Enable = FALSE;
			}
			else if(inst->Update){
				inst->Valid = FALSE;
				inst->Update = FALSE;
				inst->Internal.State = trkPAPER_SH_CLICK_INFO_LOOKUP;
				inst->Internal.Fbs.ShReadInfo.Enable = FALSE;
				inst->ErrorID = trkPAPER_SH_INFO_ERR_OK;
			}
			else if (inst->Internal.Fbs.ShReadInfo.Error) {
				inst->Valid = FALSE;
				inst->ErrorID = trkPAPER_SH_INFO_WRN_BAD_SH_READ;
			}
			else if(inst->Internal.Fbs.ShReadInfo.Valid){
				inst->Valid = TRUE;
				inst->Data.ShInfo = inst->Internal.Fbs.ShReadInfo.ShuttleInfo;
			}
			break;

		case trkPAPER_SH_BUILD_TABLE:
			//Initialize Table
			brsmemset((uintptr_t)&inst->Internal.Axes, 0, sizeof(inst->Internal.Axes));
			inst->Internal.ShuttleCount = 0;
			inst->Internal.Fbs.AsmGetShuttle.Enable = TRUE;

			inst->Internal.State = trkPAPER_SH_CLICK_GET_SH;
			break;

		case trkPAPER_SH_CLICK_GET_SH:
			//******************************************************************************** Get Shuttle state
			if(inst->Internal.Fbs.AsmGetShuttle.Error){
				inst->Error = TRUE;
				inst->ErrorID = trkPAPER_SH_INFO_ERR_INVALID_ASM;

				inst->Internal.State = trkPAPER_SH_CLICK_INFO_ERROR;
			}
			else if(inst->Internal.Fbs.AsmGetShuttle.Valid){
				if(inst->Internal.Fbs.AsmGetShuttle.TotalCount >= trkPAPER_MAX_SHUTTLE_COUNT ){
					inst->Error = TRUE;
					inst->ErrorID = trkPAPER_SH_INFO_ERR_SH_CNT_EXCD;
					inst->Internal.State = trkPAPER_SH_CLICK_INFO_ERROR;
				}
				//Populate Axes table for shuttle
				inst->Internal.Axes[inst->Internal.ShuttleCount].Present = TRUE;
				inst->Internal.Axes[inst->Internal.ShuttleCount].Axis = inst->Internal.Fbs.AsmGetShuttle.Axis;
				inst->Internal.Axes[inst->Internal.ShuttleCount].ShuttleID = inst->Internal.Fbs.AsmGetShuttle.AdditionalInfo.ShuttleID;
				inst->Internal.Fbs.AsmGetShuttle.Next = FALSE;
				inst->Internal.ShuttleCount++;

				if(inst->Internal.Fbs.AsmGetShuttle.RemainingCount == 0 ){
					//Done populating the lookup table, moving on
					inst->Internal.Fbs.AsmGetShuttle.Enable = FALSE;
					if (inst->Internal.UpdateLookupTable ) {
						inst->Internal.State =trkPAPER_SH_CLICK_INFO_LOOKUP;
						inst->ErrorID = trkPAPER_SH_INFO_ERR_OK;
						inst->Internal.UpdateLookupTable = FALSE;
					}
					else{
						inst->Internal.State = trkPAPER_SH_CLICK_INFO_RUN;
					}
				}
				else{
					//move to next shuttle
					inst->Internal.State = trkPAPER_SH_CLICK_GET_NEXT;
				}
			}

			break;

		case trkPAPER_SH_CLICK_GET_NEXT:
			//******************************************************************************** Get next shuttle state
			inst->Internal.Fbs.AsmGetShuttle.Next = TRUE;
			inst->Internal.State = trkPAPER_SH_CLICK_GET_SH;
			break;

		case trkPAPER_SH_CLICK_INFO_LOOKUP:

			//Shuttle Lookup
			inst->Internal.UpdateLookupTable = ShuttleLookup(inst->Internal.Axes, inst->Ident, &inst->Data, &inst->Internal.Fbs.ShReadInfo);

			/*remake table if shuttle is not found*/
			if(inst->Internal.UpdateLookupTable){
				inst->Internal.State = trkPAPER_SH_BUILD_TABLE;
			}
			else{
				inst->Internal.Fbs.ShReadInfo.Enable = TRUE;
				inst->Internal.State = trkPAPER_SH_CLICK_INFO_RUN;
			}
			break;

		case trkPAPER_SH_CLICK_INFO_RESET:
			inst->Error = FALSE;
			inst->ErrorID = trkPAPER_SH_INFO_ERR_OK;

			//Reset FUBs
			inst->Internal.Fbs.AsmGetShuttle.Enable = FALSE;
			inst->Internal.Fbs.ShReadInfo.Enable = FALSE;

			inst->Internal.State = trkPAPER_SH_CLICK_INFO_OFF;
			break;

		case trkPAPER_SH_CLICK_INFO_ERROR:
			if(inst->ErrorReset){
				inst->Internal.State = trkPAPER_SH_CLICK_INFO_RESET;
			}
			break;
	}
	//FB calls
	MC_BR_AsmGetShuttle_AcpTrak(&inst->Internal.Fbs.AsmGetShuttle);
	MC_BR_ShReadInfo_AcpTrak(&inst->Internal.Fbs.ShReadInfo);
}
```

### Library Logical/Libraries/AdvIecChk (IEC, version 2.00.0) - IEC Check w/ Advanced Debugging Data
Depends on: Sys_Lib, AsString

#### AdvIecChk.fun - Exported functions and function blocks
```iecst
(********************************************************************
 * COPYRIGHT --
 ********************************************************************
 * Library: IecCheck
 * File: IecCheck.fun
 * Author: adamsm
 * Created: October 03, 2012
 ********************************************************************
 * Functions and function blocks of library IecCheck
 ********************************************************************)

FUNCTION CheckDivDWord : UDINT (* Check divisor for DINT and UDINT division *)
	VAR_INPUT
		divisor : UDINT;
	END_VAR
END_FUNCTION

FUNCTION CheckDivWord : UINT (* Check divisor for INT and UINT division *)
	VAR_INPUT
		divisor : UINT;
	END_VAR
END_FUNCTION

FUNCTION CheckDivByte : USINT (* Check divisor for SINT and USINT division *)
	VAR_INPUT
		divisor : USINT;
	END_VAR
END_FUNCTION

FUNCTION CheckDivReal : REAL (* Check divisor for REAL division *)
	VAR_INPUT
		divisor : REAL;
	END_VAR
END_FUNCTION

FUNCTION CheckDivLReal : LREAL (* Check divisor for LREAL division, not available for SG3 and SGC *)
	VAR_INPUT
		divisor : LREAL;
	END_VAR
END_FUNCTION

FUNCTION CheckBounds : DINT (* Check range for array access *)
	VAR_INPUT
		index : DINT;
		lower : DINT;
		upper : DINT;
	END_VAR
	VAR
		LowString : STRING[4];
		UpString : STRING[4];
		IndexString : STRING[4];
		text : STRING[80];
	END_VAR
END_FUNCTION

FUNCTION CheckRange : DINT (* Check range for enumeration *)
	VAR_INPUT
		value : DINT;
		lower : DINT;
		upper : DINT;
	END_VAR
	VAR
		LowString : STRING[4];
		UpString : STRING[4];
		IndexString : STRING[4];
		text : STRING[80];
	END_VAR
END_FUNCTION

FUNCTION CheckSignedSubrange : DINT (* Check range for subrange of signed data types *)
	VAR_INPUT
		value : DINT;
		lower : DINT;
		upper : DINT;
	END_VAR
	VAR
		text : STRING[80];
		LowString : STRING[4];
		UpString : STRING[4];
		IndexString : STRING[4];
	END_VAR
END_FUNCTION

FUNCTION CheckUnsignedSubrange : UDINT (* Check range for subrange of unsigned data types *)
	VAR_INPUT
		value : UDINT;
		lower : UDINT;
		upper : UDINT;
	END_VAR
	VAR
		LowString : STRING[4];
		UpString : STRING[4];
		IndexString : STRING[4];
		text : STRING[80];
	END_VAR
END_FUNCTION

FUNCTION CheckReadAccess : UDINT (* Check address when reading dynamic variables *)
	VAR_INPUT
		address : UDINT;
	END_VAR
END_FUNCTION

FUNCTION CheckWriteAccess : UDINT (* Check address when writing dynamic variables *)
	VAR_INPUT
		address : UDINT;
	END_VAR
END_FUNCTION

FUNCTION MakeEntry : UDINT (* Makes an entry (log book entry) in the error log book *)
	VAR_INPUT
		number : UINT;
		index : DINT;
		text : STRING[80];
	END_VAR
	VAR
		taskname : STRING[30];
		group : USINT;
		status_name : UINT;
		out_text : STRING[190];
		pv_adr : UDINT;
		data_len : UDINT;
		SectionString : STRING[80];
		SectionData : DINT;
	END_VAR
END_FUNCTION
```
